FUNCTION_BLOCK "ifbHMISelectBLK"
{ S7_Optimized_Access := 'TRUE' }
VERSION : 0.1
   VAR
      edge : Array[0..50] of Bool;
   END_VAR

   VAR_TEMP
      blockSelected : Int;
      arrChildIndex : Array[0..50] of Int;
      tempEdge : Bool;
   END_VAR


BEGIN
NETWORK
TITLE = Get the selected BLK
//------------------------------------------------------------------------//
// Get the BLK index number selected by the user when they clicked the    //
// faceplate BLK target:                                                  //
//------------------------------------------------------------------------//
      L "dbHMIInterfaceBLK".block.blockSelected;
      T #blockSelected;

NETWORK
TITLE =
      A(;
      L #blockSelected;
      L 1134;
      ==I;
      );
      FP #edge[0];
      = #tempEdge;
      JCN out1;

      A "idbEMA1".f[0].p.read.mc.modeAUTO;
      R "dbHMIInterfaceBLK".block.manual;

      A "idbEMA1".f[0].p.read.mc.modeMANUAL;
      S "dbHMIInterfaceBLK".block.manual;

out1:      NOP 0;

NETWORK
TITLE = EA1010 M1 Vessel Agitator
//------------------------------------------------------------------------//
// Check if this BLK instance is selected:                                //
//------------------------------------------------------------------------//
      A(;
      L #blockSelected;
      L 1134;
      ==I;
      );

      JCN _not_EA1010;
      AN #tempEdge;
      CALL "fcHMIInterfaceBLK"
      (  mcr                         := "idbEMA1".f[0].p.read.mc ,
         mcw                         := "idbEMA1".f[0].p.write.mc ,
         bmc                         := "idbEMA1".f[0].p.read.bmc
      );

NETWORK
TITLE = Transfer the child state values and errors to the interface array
//------------------------------------------------------------------------//
// Transfer the child states and if they have any error condition:        //
//------------------------------------------------------------------------//
      L 0        ;// SIC_AGIT SIC1
      T #arrChildIndex[1];
      L "idbSIC1".f[#arrChildIndex[1]].p.read.mc.STATE;
      T "dbHMIInterfaceBLK".block.arrChildState[1];
      A "idbSIC1".f[#arrChildIndex[1]].p.read.mc.ERROR;
      = "dbHMIInterfaceBLK".block.arrChildError[1];
      A "idbSIC1".f[#arrChildIndex[1]].p.read.mc.INTERLOCK;
      = "dbHMIInterfaceBLK".block.arrChildInterlock[1];

NETWORK
TITLE = Transfer the parameter values to the interface arrays
//------------------------------------------------------------------------//
// Transfer the parameter values:                                         //
//------------------------------------------------------------------------//
      AN "dbHMIInterfaceBLK".block.manual;
      JCN _manual_EA1010;
      A "idbEMA1".f[0].p.read.AGIT_RUNNING;
      = "dbHMIInterfaceBLK".block.arrBool[1];
      A "idbEMA1".f[0].p.read.AGIT_STOPPED;
      = "dbHMIInterfaceBLK".block.arrBool[2];
      A "idbEMA1".f[0].p.read.RESETRUNTIMER;
      = "dbHMIInterfaceBLK".block.arrBool[3];
      L "idbEMA1".f[0].p.read.ACUMTIMEH;
      T "dbHMIInterfaceBLK".block.arrInt[1];
      L "idbEMA1".f[0].p.read.ACUMTIMEM;
      T "dbHMIInterfaceBLK".block.arrInt[2];
      L "idbEMA1".f[0].p.read.ACUMTIMES;
      T "dbHMIInterfaceBLK".block.arrInt[3];
      L "idbEMA1".f[0].p.write.RUNTIME_H;
      T "dbHMIInterfaceBLK".block.arrInt[4];
      L "idbEMA1".f[0].p.write.RUNTIME_M;
      T "dbHMIInterfaceBLK".block.arrInt[5];
      L "idbEMA1".f[0].p.write.RUNTIME_S;
      T "dbHMIInterfaceBLK".block.arrInt[6];
      L "idbEMA1".f[0].p.write.SETPOINT;
      T "dbHMIInterfaceBLK".block.arrReal[1];
_manual_EA1010:      NOP 0;

NETWORK
TITLE = Transfer the parameter values to the interface arrays
//------------------------------------------------------------------------//
// Transfer the parameter values:                                         //
//------------------------------------------------------------------------//
      A "dbHMIInterfaceBLK".block.manual;
      JCN _auto_EA1010;
      A "dbHMIInterfaceBLK".block.arrBool[1];
      = "idbEMA1".f[0].p.read.AGIT_RUNNING;
      A "dbHMIInterfaceBLK".block.arrBool[2];
      = "idbEMA1".f[0].p.read.AGIT_STOPPED;
      A "dbHMIInterfaceBLK".block.arrBool[3];
      = "idbEMA1".f[0].p.read.RESETRUNTIMER;
      L "dbHMIInterfaceBLK".block.arrInt[1];
      T "idbEMA1".f[0].p.read.ACUMTIMEH;
      L "dbHMIInterfaceBLK".block.arrInt[2];
      T "idbEMA1".f[0].p.read.ACUMTIMEM;
      L "dbHMIInterfaceBLK".block.arrInt[3];
      T "idbEMA1".f[0].p.read.ACUMTIMES;
      L "dbHMIInterfaceBLK".block.arrInt[4];
      T "idbEMA1".f[0].p.write.RUNTIME_H;
      L "dbHMIInterfaceBLK".block.arrInt[5];
      T "idbEMA1".f[0].p.write.RUNTIME_M;
      L "dbHMIInterfaceBLK".block.arrInt[6];
      T "idbEMA1".f[0].p.write.RUNTIME_S;
      L "dbHMIInterfaceBLK".block.arrReal[1];
      T "idbEMA1".f[0].p.write.SETPOINT;
_auto_EA1010:      NOP 0;

_not_EA1010:      NOP 0;

NETWORK
TITLE = EC1001 M1 LP CA and HP CA supply and Vacuum and Vent
//------------------------------------------------------------------------//
// Check if this BLK instance is selected:                                //
//------------------------------------------------------------------------//
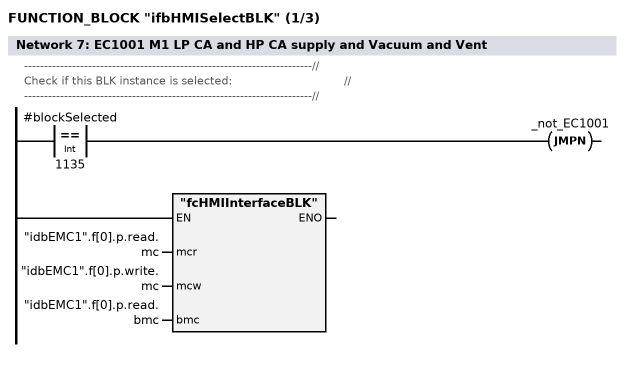
      A(;
      L #blockSelected;
      L 1135;
      ==I;
      );
      JCN _not_EC1001;

      CALL "fcHMIInterfaceBLK"
      (  mcr                         := "idbEMC1".f[0].p.read.mc ,
         mcw                         := "idbEMC1".f[0].p.write.mc ,
         bmc                         := "idbEMC1".f[0].p.read.bmc
      );

NETWORK
TITLE = Transfer the child state values and errors to the interface array
//------------------------------------------------------------------------//
// Transfer the child states and if they have any error condition:        //
//------------------------------------------------------------------------//
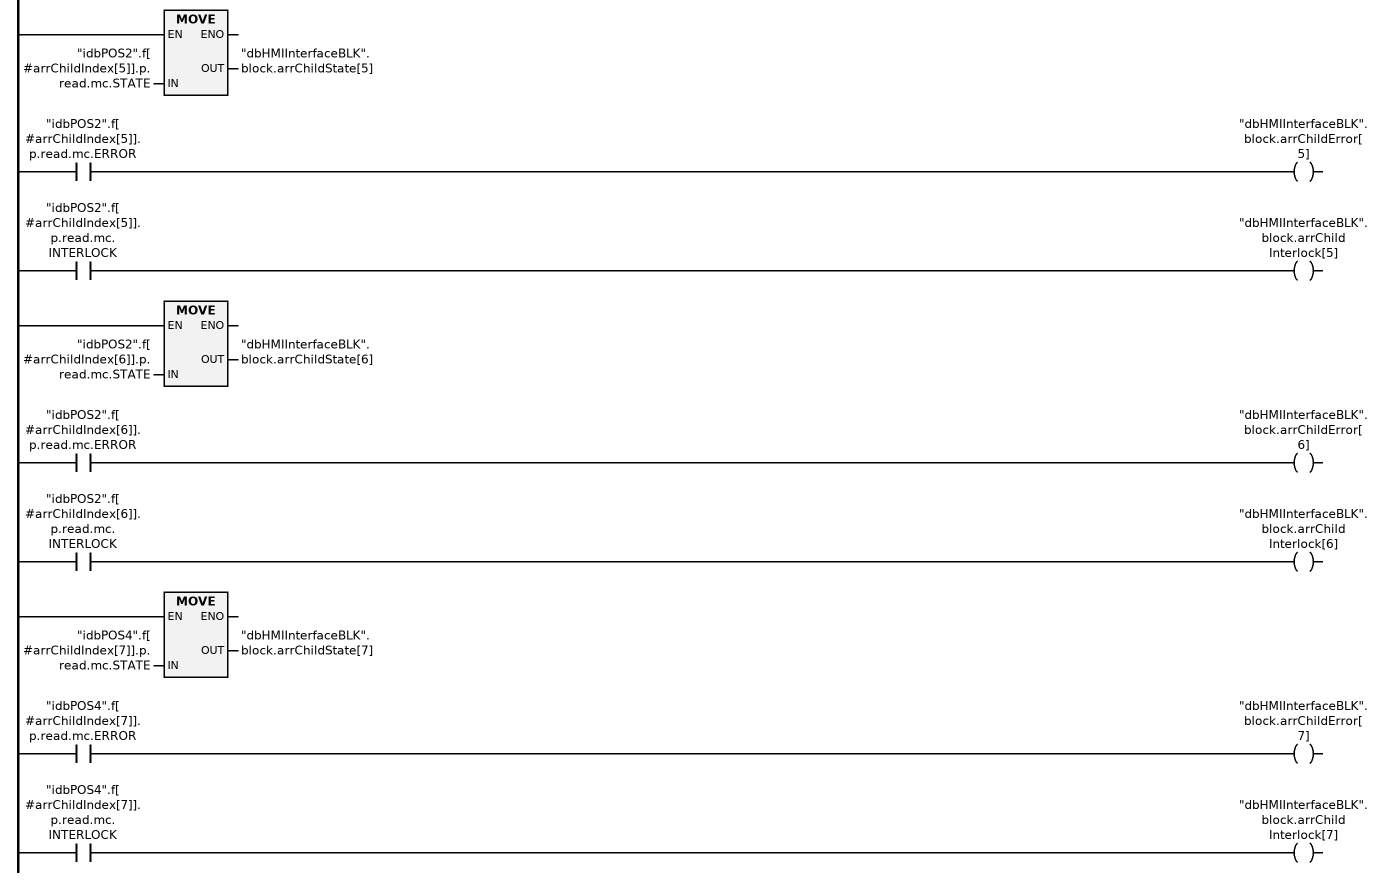
      L 0        ;// PC_VESSEL PC1
      T #arrChildIndex[1];
      L 0        ;// PI_VESSEL PI1
      T #arrChildIndex[2];
      L 1        ;// POS_HPCA POS2
      T #arrChildIndex[3];
      L 2        ;// POS_LPCA POS2
      T #arrChildIndex[4];
      L 3        ;// POS_VACUUM POS2
      T #arrChildIndex[5];
      L 0        ;// POS_VENT POS2
      T #arrChildIndex[6];
      L 0        ;// POS_DRAIN POS4
      T #arrChildIndex[7];
      L "idbPC1".f[#arrChildIndex[1]].p.read.mc.STATE;
      T "dbHMIInterfaceBLK".block.arrChildState[1];
      A "idbPC1".f[#arrChildIndex[1]].p.read.mc.ERROR;
      = "dbHMIInterfaceBLK".block.arrChildError[1];
      A "idbPC1".f[#arrChildIndex[1]].p.read.mc.INTERLOCK;
      = "dbHMIInterfaceBLK".block.arrChildInterlock[1];
      L "idbPI1".f[#arrChildIndex[2]].p.read.mc.STATE;
      T "dbHMIInterfaceBLK".block.arrChildState[2];
      A "idbPI1".f[#arrChildIndex[2]].p.read.mc.ERROR;
      = "dbHMIInterfaceBLK".block.arrChildError[2];
      A "idbPI1".f[#arrChildIndex[2]].p.read.mc.INTERLOCK;
      = "dbHMIInterfaceBLK".block.arrChildInterlock[2];
      L "idbPOS2".f[#arrChildIndex[3]].p.read.mc.STATE;
      T "dbHMIInterfaceBLK".block.arrChildState[3];
      A "idbPOS2".f[#arrChildIndex[3]].p.read.mc.ERROR;
      = "dbHMIInterfaceBLK".block.arrChildError[3];
      A "idbPOS2".f[#arrChildIndex[3]].p.read.mc.INTERLOCK;
      = "dbHMIInterfaceBLK".block.arrChildInterlock[3];
      L "idbPOS2".f[#arrChildIndex[4]].p.read.mc.STATE;
      T "dbHMIInterfaceBLK".block.arrChildState[4];
      A "idbPOS2".f[#arrChildIndex[4]].p.read.mc.ERROR;
      = "dbHMIInterfaceBLK".block.arrChildError[4];
      A "idbPOS2".f[#arrChildIndex[4]].p.read.mc.INTERLOCK;
      = "dbHMIInterfaceBLK".block.arrChildInterlock[4];
      L "idbPOS2".f[#arrChildIndex[5]].p.read.mc.STATE;
      T "dbHMIInterfaceBLK".block.arrChildState[5];
      A "idbPOS2".f[#arrChildIndex[5]].p.read.mc.ERROR;
      = "dbHMIInterfaceBLK".block.arrChildError[5];
      A "idbPOS2".f[#arrChildIndex[5]].p.read.mc.INTERLOCK;
      = "dbHMIInterfaceBLK".block.arrChildInterlock[5];
      L "idbPOS2".f[#arrChildIndex[6]].p.read.mc.STATE;
      T "dbHMIInterfaceBLK".block.arrChildState[6];
      A "idbPOS2".f[#arrChildIndex[6]].p.read.mc.ERROR;
      = "dbHMIInterfaceBLK".block.arrChildError[6];
      A "idbPOS2".f[#arrChildIndex[6]].p.read.mc.INTERLOCK;
      = "dbHMIInterfaceBLK".block.arrChildInterlock[6];
      L "idbPOS4".f[#arrChildIndex[7]].p.read.mc.STATE;
      T "dbHMIInterfaceBLK".block.arrChildState[7];
      A "idbPOS4".f[#arrChildIndex[7]].p.read.mc.ERROR;
      = "dbHMIInterfaceBLK".block.arrChildError[7];
      A "idbPOS4".f[#arrChildIndex[7]].p.read.mc.INTERLOCK;
      = "dbHMIInterfaceBLK".block.arrChildInterlock[7];

NETWORK
TITLE = Transfer the parameter values to the interface arrays
//------------------------------------------------------------------------//
// Transfer the parameter values:                                         //
//------------------------------------------------------------------------//
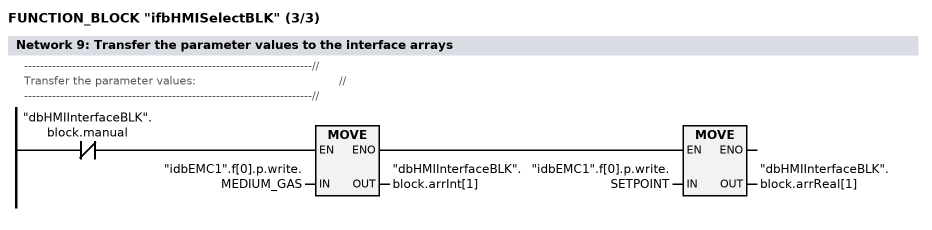
      AN "dbHMIInterfaceBLK".block.manual;
      JCN _manual_EC1001;
      L "idbEMC1".f[0].p.write.MEDIUM_GAS;
      T "dbHMIInterfaceBLK".block.arrInt[1];
      L "idbEMC1".f[0].p.write.SETPOINT;
      T "dbHMIInterfaceBLK".block.arrReal[1];
_manual_EC1001:      NOP 0;

NETWORK
TITLE = Transfer the parameter values to the interface arrays
//------------------------------------------------------------------------//
// Transfer the parameter values:                                         //
//------------------------------------------------------------------------//
      A "dbHMIInterfaceBLK".block.manual;
      JCN _auto_EC1001;
      L "dbHMIInterfaceBLK".block.arrInt[1];
      T "idbEMC1".f[0].p.write.MEDIUM_GAS;
      L "dbHMIInterfaceBLK".block.arrReal[1];
      T "idbEMC1".f[0].p.write.SETPOINT;
_auto_EC1001:      NOP 0;

_not_EC1001:      NOP 0;

NETWORK
TITLE = EC1002 M1 WFI and PS supply plus PW and PS supply
//------------------------------------------------------------------------//
// Check if this BLK instance is selected:                                //
//------------------------------------------------------------------------//
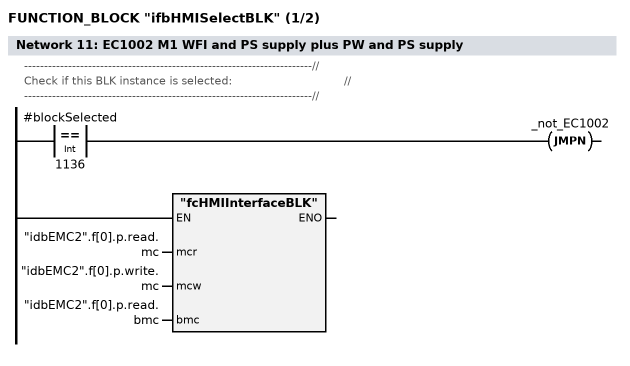
      A(;
      L #blockSelected;
      L 1136;
      ==I;
      );
      JCN _not_EC1002;

      CALL "fcHMIInterfaceBLK"
      (  mcr                         := "idbEMC2".f[0].p.read.mc ,
         mcw                         := "idbEMC2".f[0].p.write.mc ,
         bmc                         := "idbEMC2".f[0].p.read.bmc
      );

NETWORK
TITLE = Transfer the child state values and errors to the interface array
//------------------------------------------------------------------------//
// Transfer the child states and if they have any error condition:        //
//------------------------------------------------------------------------//
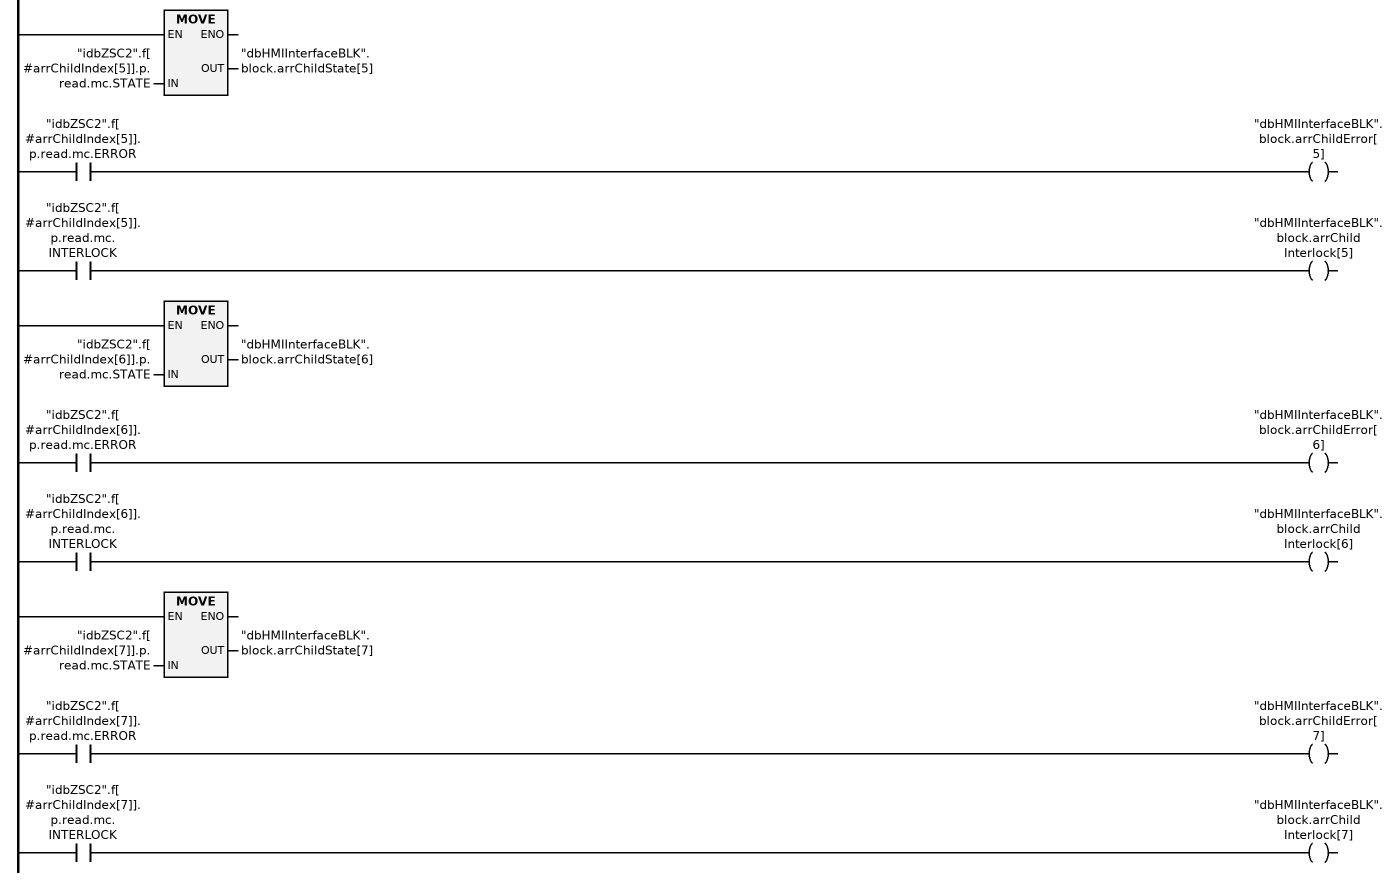
      L 5        ;// POS_PSPW POS2
      T #arrChildIndex[1];
      L 4        ;// POS_PSWFI POS2
      T #arrChildIndex[2];
      L 29        ;// POS_PW POS4
      T #arrChildIndex[3];
      L 28        ;// POS_WFI POS4
      T #arrChildIndex[4];
      L 2        ;// ZSC_FPINLET ZSC2
      T #arrChildIndex[5];
      L 1        ;// ZSC_FPPW ZSC2
      T #arrChildIndex[6];
      L 0        ;// ZSC_FPWFI ZSC2
      T #arrChildIndex[7];
      L "idbPOS2".f[#arrChildIndex[1]].p.read.mc.STATE;
      T "dbHMIInterfaceBLK".block.arrChildState[1];
      A "idbPOS2".f[#arrChildIndex[1]].p.read.mc.ERROR;
      = "dbHMIInterfaceBLK".block.arrChildError[1];
      A "idbPOS2".f[#arrChildIndex[1]].p.read.mc.INTERLOCK;
      = "dbHMIInterfaceBLK".block.arrChildInterlock[1];
      L "idbPOS2".f[#arrChildIndex[2]].p.read.mc.STATE;
      T "dbHMIInterfaceBLK".block.arrChildState[2];
      A "idbPOS2".f[#arrChildIndex[2]].p.read.mc.ERROR;
      = "dbHMIInterfaceBLK".block.arrChildError[2];
      A "idbPOS2".f[#arrChildIndex[2]].p.read.mc.INTERLOCK;
      = "dbHMIInterfaceBLK".block.arrChildInterlock[2];
      L "idbPOS4".f[#arrChildIndex[3]].p.read.mc.STATE;
      T "dbHMIInterfaceBLK".block.arrChildState[3];
      A "idbPOS4".f[#arrChildIndex[3]].p.read.mc.ERROR;
      = "dbHMIInterfaceBLK".block.arrChildError[3];
      A "idbPOS4".f[#arrChildIndex[3]].p.read.mc.INTERLOCK;
      = "dbHMIInterfaceBLK".block.arrChildInterlock[3];
      L "idbPOS4".f[#arrChildIndex[4]].p.read.mc.STATE;
      T "dbHMIInterfaceBLK".block.arrChildState[4];
      A "idbPOS4".f[#arrChildIndex[4]].p.read.mc.ERROR;
      = "dbHMIInterfaceBLK".block.arrChildError[4];
      A "idbPOS4".f[#arrChildIndex[4]].p.read.mc.INTERLOCK;
      = "dbHMIInterfaceBLK".block.arrChildInterlock[4];
      L "idbZSC2".f[#arrChildIndex[5]].p.read.mc.STATE;
      T "dbHMIInterfaceBLK".block.arrChildState[5];
      A "idbZSC2".f[#arrChildIndex[5]].p.read.mc.ERROR;
      = "dbHMIInterfaceBLK".block.arrChildError[5];
      A "idbZSC2".f[#arrChildIndex[5]].p.read.mc.INTERLOCK;
      = "dbHMIInterfaceBLK".block.arrChildInterlock[5];
      L "idbZSC2".f[#arrChildIndex[6]].p.read.mc.STATE;
      T "dbHMIInterfaceBLK".block.arrChildState[6];
      A "idbZSC2".f[#arrChildIndex[6]].p.read.mc.ERROR;
      = "dbHMIInterfaceBLK".block.arrChildError[6];
      A "idbZSC2".f[#arrChildIndex[6]].p.read.mc.INTERLOCK;
      = "dbHMIInterfaceBLK".block.arrChildInterlock[6];
      L "idbZSC2".f[#arrChildIndex[7]].p.read.mc.STATE;
      T "dbHMIInterfaceBLK".block.arrChildState[7];
      A "idbZSC2".f[#arrChildIndex[7]].p.read.mc.ERROR;
      = "dbHMIInterfaceBLK".block.arrChildError[7];
      A "idbZSC2".f[#arrChildIndex[7]].p.read.mc.INTERLOCK;
      = "dbHMIInterfaceBLK".block.arrChildInterlock[7];

NETWORK
TITLE = Transfer the parameter values to the interface arrays
//------------------------------------------------------------------------//
// Transfer the parameter values:                                         //
//------------------------------------------------------------------------//
      AN "dbHMIInterfaceBLK".block.manual;
      JCN _manual_EC1002;
      A "idbEMC2".f[0].p.read.MASS_READY;
      = "dbHMIInterfaceBLK".block.arrBool[1];
      L "idbEMC2".f[0].p.write.MEDIUM_LIQUID;
      T "dbHMIInterfaceBLK".block.arrInt[1];
      L "idbEMC2".f[0].p.read.MASS_ACTUAL;
      T "dbHMIInterfaceBLK".block.arrReal[1];
      L "idbEMC2".f[0].p.read.MASS_FINAL;
      T "dbHMIInterfaceBLK".block.arrReal[2];
      L "idbEMC2".f[0].p.read.MASS_INITIAL;
      T "dbHMIInterfaceBLK".block.arrReal[3];
      L "idbEMC2".f[0].p.write.MASS_CHARGE;
      T "dbHMIInterfaceBLK".block.arrReal[4];
      L "idbEMC2".f[0].p.write.RUNTIME;
      T "dbHMIInterfaceBLK".block.arrTime[1];
      L "idbEMC2".f[0].p.write.TIMEOUT;
      T "dbHMIInterfaceBLK".block.arrTime[2];
_manual_EC1002:      NOP 0;

NETWORK
TITLE = Transfer the parameter values to the interface arrays
//------------------------------------------------------------------------//
// Transfer the parameter values:                                         //
//------------------------------------------------------------------------//
      A "dbHMIInterfaceBLK".block.manual;
      JCN _auto_EC1002;
      A "dbHMIInterfaceBLK".block.arrBool[1];
      = "idbEMC2".f[0].p.read.MASS_READY;
      L "dbHMIInterfaceBLK".block.arrInt[1];
      T "idbEMC2".f[0].p.write.MEDIUM_LIQUID;
      L "dbHMIInterfaceBLK".block.arrReal[1];
      T "idbEMC2".f[0].p.read.MASS_ACTUAL;
      L "dbHMIInterfaceBLK".block.arrReal[2];
      T "idbEMC2".f[0].p.read.MASS_FINAL;
      L "dbHMIInterfaceBLK".block.arrReal[3];
      T "idbEMC2".f[0].p.read.MASS_INITIAL;
      L "dbHMIInterfaceBLK".block.arrReal[4];
      T "idbEMC2".f[0].p.write.MASS_CHARGE;
      L "dbHMIInterfaceBLK".block.arrTime[1];
      T "idbEMC2".f[0].p.write.RUNTIME;
      L "dbHMIInterfaceBLK".block.arrTime[2];
      T "idbEMC2".f[0].p.write.TIMEOUT;
_auto_EC1002:      NOP 0;

_not_EC1002:      NOP 0;

NETWORK
TITLE = EC3001 S1 LP CA and HP CA supply and Vacuum and Vent
//------------------------------------------------------------------------//
// Check if this BLK instance is selected:                                //
//------------------------------------------------------------------------//
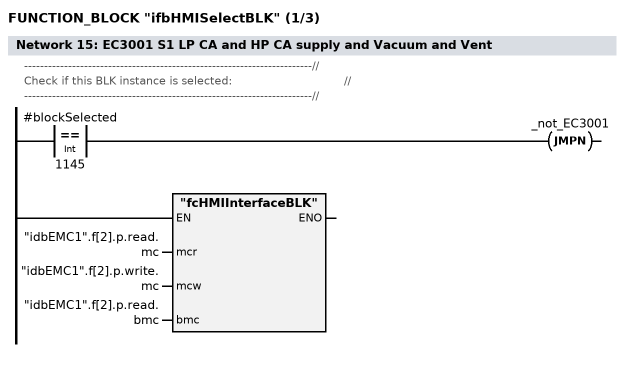
      A(;
      L #blockSelected;
      L 1145;
      ==I;
      );
      JCN _not_EC3001;

      CALL "fcHMIInterfaceBLK"
      (  mcr                         := "idbEMC1".f[2].p.read.mc ,
         mcw                         := "idbEMC1".f[2].p.write.mc ,
         bmc                         := "idbEMC1".f[2].p.read.bmc
      );

NETWORK
TITLE = Transfer the child state values and errors to the interface array
//------------------------------------------------------------------------//
// Transfer the child states and if they have any error condition:        //
//------------------------------------------------------------------------//
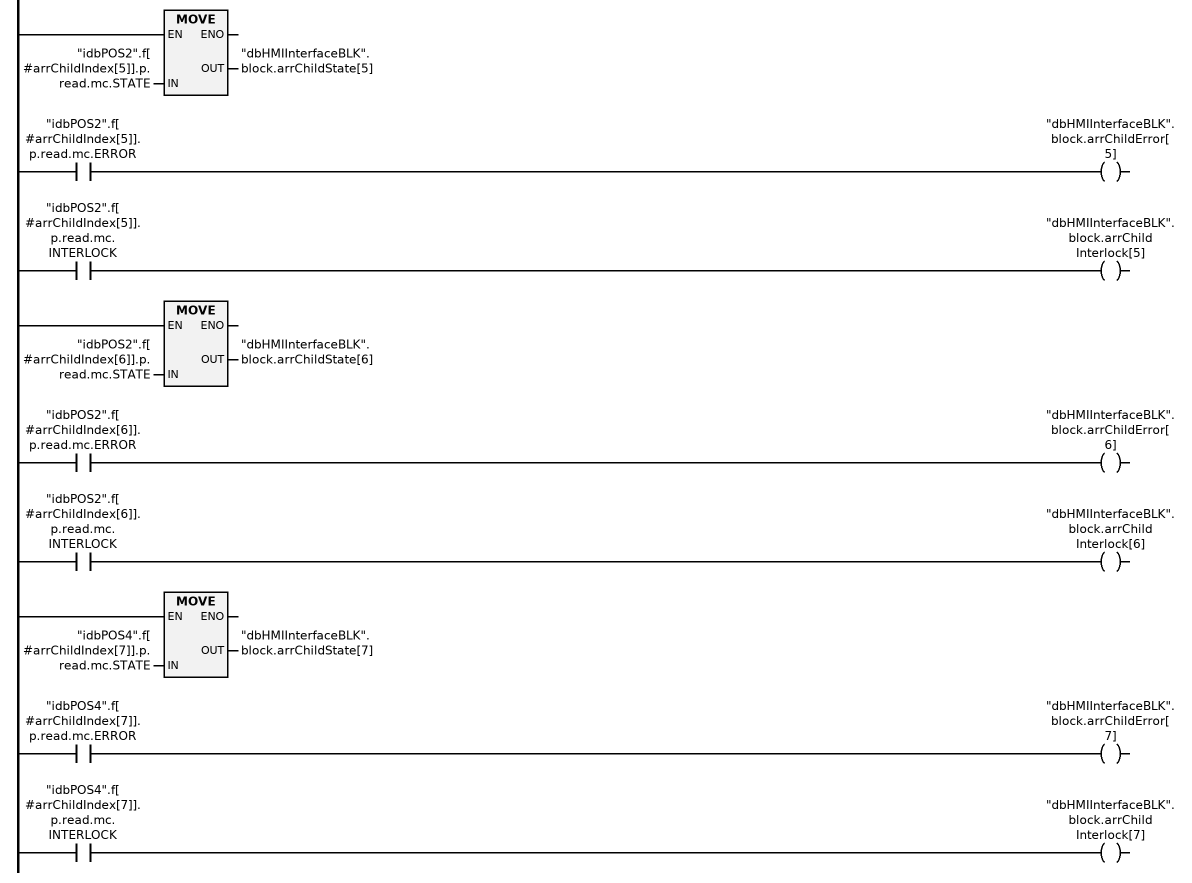
      L 2        ;// PC_VESSEL PC1
      T #arrChildIndex[1];
      L 2        ;// PI_VESSEL PI1
      T #arrChildIndex[2];
      L 27        ;// POS_HPCA POS2
      T #arrChildIndex[3];
      L 28        ;// POS_LPCA POS2
      T #arrChildIndex[4];
      L 29        ;// POS_VACUUM POS2
      T #arrChildIndex[5];
      L 26        ;// POS_VENT POS2
      T #arrChildIndex[6];
      L 16        ;// POS_DRAIN POS4
      T #arrChildIndex[7];
      L "idbPC1".f[#arrChildIndex[1]].p.read.mc.STATE;
      T "dbHMIInterfaceBLK".block.arrChildState[1];
      A "idbPC1".f[#arrChildIndex[1]].p.read.mc.ERROR;
      = "dbHMIInterfaceBLK".block.arrChildError[1];
      A "idbPC1".f[#arrChildIndex[1]].p.read.mc.INTERLOCK;
      = "dbHMIInterfaceBLK".block.arrChildInterlock[1];
      L "idbPI1".f[#arrChildIndex[2]].p.read.mc.STATE;
      T "dbHMIInterfaceBLK".block.arrChildState[2];
      A "idbPI1".f[#arrChildIndex[2]].p.read.mc.ERROR;
      = "dbHMIInterfaceBLK".block.arrChildError[2];
      A "idbPI1".f[#arrChildIndex[2]].p.read.mc.INTERLOCK;
      = "dbHMIInterfaceBLK".block.arrChildInterlock[2];
      L "idbPOS2".f[#arrChildIndex[3]].p.read.mc.STATE;
      T "dbHMIInterfaceBLK".block.arrChildState[3];
      A "idbPOS2".f[#arrChildIndex[3]].p.read.mc.ERROR;
      = "dbHMIInterfaceBLK".block.arrChildError[3];
      A "idbPOS2".f[#arrChildIndex[3]].p.read.mc.INTERLOCK;
      = "dbHMIInterfaceBLK".block.arrChildInterlock[3];
      L "idbPOS2".f[#arrChildIndex[4]].p.read.mc.STATE;
      T "dbHMIInterfaceBLK".block.arrChildState[4];
      A "idbPOS2".f[#arrChildIndex[4]].p.read.mc.ERROR;
      = "dbHMIInterfaceBLK".block.arrChildError[4];
      A "idbPOS2".f[#arrChildIndex[4]].p.read.mc.INTERLOCK;
      = "dbHMIInterfaceBLK".block.arrChildInterlock[4];
      L "idbPOS2".f[#arrChildIndex[5]].p.read.mc.STATE;
      T "dbHMIInterfaceBLK".block.arrChildState[5];
      A "idbPOS2".f[#arrChildIndex[5]].p.read.mc.ERROR;
      = "dbHMIInterfaceBLK".block.arrChildError[5];
      A "idbPOS2".f[#arrChildIndex[5]].p.read.mc.INTERLOCK;
      = "dbHMIInterfaceBLK".block.arrChildInterlock[5];
      L "idbPOS2".f[#arrChildIndex[6]].p.read.mc.STATE;
      T "dbHMIInterfaceBLK".block.arrChildState[6];
      A "idbPOS2".f[#arrChildIndex[6]].p.read.mc.ERROR;
      = "dbHMIInterfaceBLK".block.arrChildError[6];
      A "idbPOS2".f[#arrChildIndex[6]].p.read.mc.INTERLOCK;
      = "dbHMIInterfaceBLK".block.arrChildInterlock[6];
      L "idbPOS4".f[#arrChildIndex[7]].p.read.mc.STATE;
      T "dbHMIInterfaceBLK".block.arrChildState[7];
      A "idbPOS4".f[#arrChildIndex[7]].p.read.mc.ERROR;
      = "dbHMIInterfaceBLK".block.arrChildError[7];
      A "idbPOS4".f[#arrChildIndex[7]].p.read.mc.INTERLOCK;
      = "dbHMIInterfaceBLK".block.arrChildInterlock[7];

NETWORK
TITLE = Transfer the parameter values to the interface arrays
//------------------------------------------------------------------------//
// Transfer the parameter values:                                         //
//------------------------------------------------------------------------//
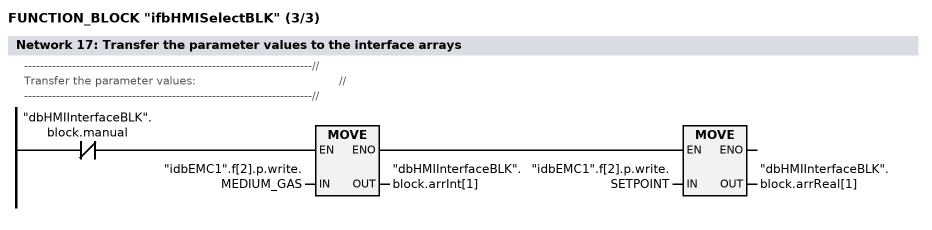
      AN "dbHMIInterfaceBLK".block.manual;
      JCN _manual_EC3001;
      L "idbEMC1".f[2].p.write.MEDIUM_GAS;
      T "dbHMIInterfaceBLK".block.arrInt[1];
      L "idbEMC1".f[2].p.write.SETPOINT;
      T "dbHMIInterfaceBLK".block.arrReal[1];
_manual_EC3001:      NOP 0;

NETWORK
TITLE = Transfer the parameter values to the interface arrays
//------------------------------------------------------------------------//
// Transfer the parameter values:                                         //
//------------------------------------------------------------------------//
      A "dbHMIInterfaceBLK".block.manual;
      JCN _auto_EC3001;
      L "dbHMIInterfaceBLK".block.arrInt[1];
      T "idbEMC1".f[2].p.write.MEDIUM_GAS;
      L "dbHMIInterfaceBLK".block.arrReal[1];
      T "idbEMC1".f[2].p.write.SETPOINT;
_auto_EC3001:      NOP 0;

_not_EC3001:      NOP 0;

NETWORK
TITLE = EC3002 S1 WFI and PS supply plus PW and PS supply
//------------------------------------------------------------------------//
// Check if this BLK instance is selected:                                //
//------------------------------------------------------------------------//
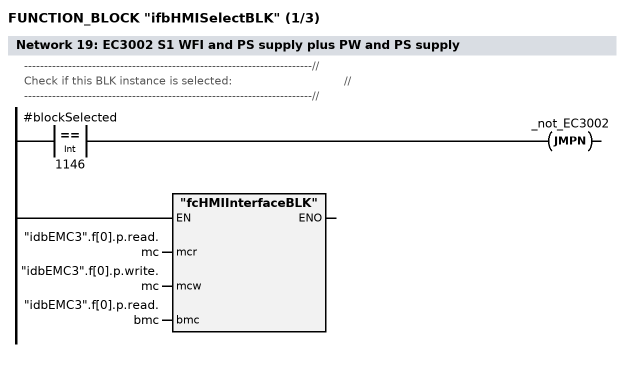
      A(;
      L #blockSelected;
      L 1146;
      ==I;
      );
      JCN _not_EC3002;

      CALL "fcHMIInterfaceBLK"
      (  mcr                         := "idbEMC3".f[0].p.read.mc ,
         mcw                         := "idbEMC3".f[0].p.write.mc ,
         bmc                         := "idbEMC3".f[0].p.read.bmc
      );

NETWORK
TITLE = Transfer the child state values and errors to the interface array
//------------------------------------------------------------------------//
// Transfer the child states and if they have any error condition:        //
//------------------------------------------------------------------------//
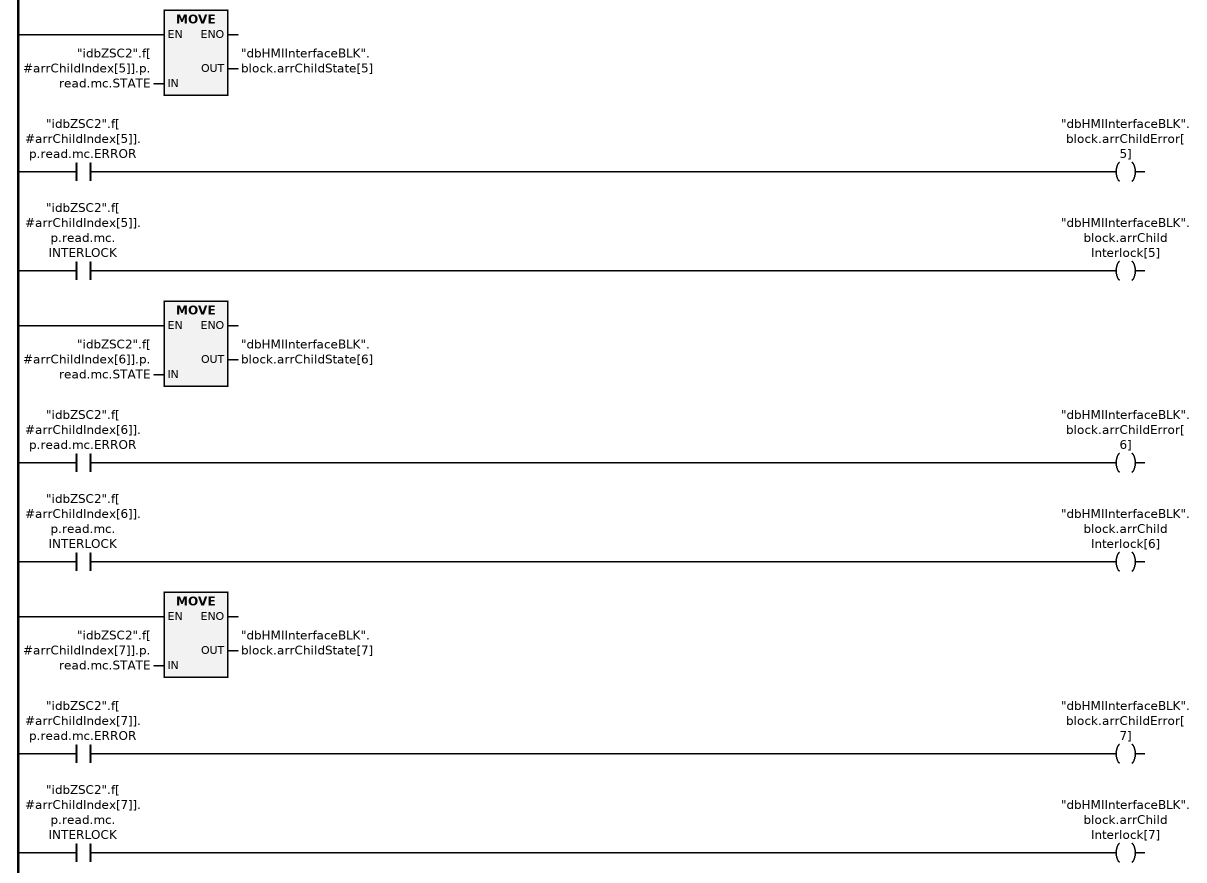
      L 31        ;// POS_PSPW POS2
      T #arrChildIndex[1];
      L 30        ;// POS_PSWFI POS2
      T #arrChildIndex[2];
      L 33        ;// POS_PW POS4
      T #arrChildIndex[3];
      L 32        ;// POS_WFI POS4
      T #arrChildIndex[4];
      L 16        ;// ZSC_FPINLET ZSC2
      T #arrChildIndex[5];
      L 15        ;// ZSC_FPPW ZSC2
      T #arrChildIndex[6];
      L 14        ;// ZSC_FPWFI ZSC2
      T #arrChildIndex[7];
      L "idbPOS2".f[#arrChildIndex[1]].p.read.mc.STATE;
      T "dbHMIInterfaceBLK".block.arrChildState[1];
      A "idbPOS2".f[#arrChildIndex[1]].p.read.mc.ERROR;
      = "dbHMIInterfaceBLK".block.arrChildError[1];
      A "idbPOS2".f[#arrChildIndex[1]].p.read.mc.INTERLOCK;
      = "dbHMIInterfaceBLK".block.arrChildInterlock[1];
      L "idbPOS2".f[#arrChildIndex[2]].p.read.mc.STATE;
      T "dbHMIInterfaceBLK".block.arrChildState[2];
      A "idbPOS2".f[#arrChildIndex[2]].p.read.mc.ERROR;
      = "dbHMIInterfaceBLK".block.arrChildError[2];
      A "idbPOS2".f[#arrChildIndex[2]].p.read.mc.INTERLOCK;
      = "dbHMIInterfaceBLK".block.arrChildInterlock[2];
      L "idbPOS4".f[#arrChildIndex[3]].p.read.mc.STATE;
      T "dbHMIInterfaceBLK".block.arrChildState[3];
      A "idbPOS4".f[#arrChildIndex[3]].p.read.mc.ERROR;
      = "dbHMIInterfaceBLK".block.arrChildError[3];
      A "idbPOS4".f[#arrChildIndex[3]].p.read.mc.INTERLOCK;
      = "dbHMIInterfaceBLK".block.arrChildInterlock[3];
      L "idbPOS4".f[#arrChildIndex[4]].p.read.mc.STATE;
      T "dbHMIInterfaceBLK".block.arrChildState[4];
      A "idbPOS4".f[#arrChildIndex[4]].p.read.mc.ERROR;
      = "dbHMIInterfaceBLK".block.arrChildError[4];
      A "idbPOS4".f[#arrChildIndex[4]].p.read.mc.INTERLOCK;
      = "dbHMIInterfaceBLK".block.arrChildInterlock[4];
      L "idbZSC2".f[#arrChildIndex[5]].p.read.mc.STATE;
      T "dbHMIInterfaceBLK".block.arrChildState[5];
      A "idbZSC2".f[#arrChildIndex[5]].p.read.mc.ERROR;
      = "dbHMIInterfaceBLK".block.arrChildError[5];
      A "idbZSC2".f[#arrChildIndex[5]].p.read.mc.INTERLOCK;
      = "dbHMIInterfaceBLK".block.arrChildInterlock[5];
      L "idbZSC2".f[#arrChildIndex[6]].p.read.mc.STATE;
      T "dbHMIInterfaceBLK".block.arrChildState[6];
      A "idbZSC2".f[#arrChildIndex[6]].p.read.mc.ERROR;
      = "dbHMIInterfaceBLK".block.arrChildError[6];
      A "idbZSC2".f[#arrChildIndex[6]].p.read.mc.INTERLOCK;
      = "dbHMIInterfaceBLK".block.arrChildInterlock[6];
      L "idbZSC2".f[#arrChildIndex[7]].p.read.mc.STATE;
      T "dbHMIInterfaceBLK".block.arrChildState[7];
      A "idbZSC2".f[#arrChildIndex[7]].p.read.mc.ERROR;
      = "dbHMIInterfaceBLK".block.arrChildError[7];
      A "idbZSC2".f[#arrChildIndex[7]].p.read.mc.INTERLOCK;
      = "dbHMIInterfaceBLK".block.arrChildInterlock[7];

NETWORK
TITLE = Transfer the parameter values to the interface arrays
//------------------------------------------------------------------------//
// Transfer the parameter values:                                         //
//------------------------------------------------------------------------//
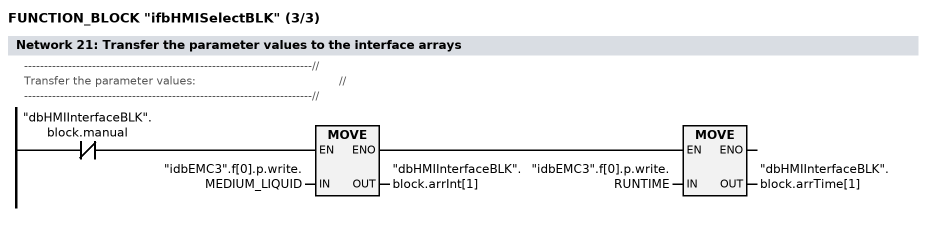
      AN "dbHMIInterfaceBLK".block.manual;
      JCN _manual_EC3002;
      L "idbEMC3".f[0].p.write.MEDIUM_LIQUID;
      T "dbHMIInterfaceBLK".block.arrInt[1];
      L "idbEMC3".f[0].p.write.RUNTIME;
      T "dbHMIInterfaceBLK".block.arrTime[1];
_manual_EC3002:      NOP 0;

NETWORK
TITLE = Transfer the parameter values to the interface arrays
//------------------------------------------------------------------------//
// Transfer the parameter values:                                         //
//------------------------------------------------------------------------//
      A "dbHMIInterfaceBLK".block.manual;
      JCN _auto_EC3002;
      L "dbHMIInterfaceBLK".block.arrInt[1];
      T "idbEMC3".f[0].p.write.MEDIUM_LIQUID;
      L "dbHMIInterfaceBLK".block.arrTime[1];
      T "idbEMC3".f[0].p.write.RUNTIME;
_auto_EC3002:      NOP 0;

_not_EC3002:      NOP 0;

NETWORK
TITLE = EG1005 M1 gas filter heating and drain valve and temperature indicator
//------------------------------------------------------------------------//
// Check if this BLK instance is selected:                                //
//------------------------------------------------------------------------//
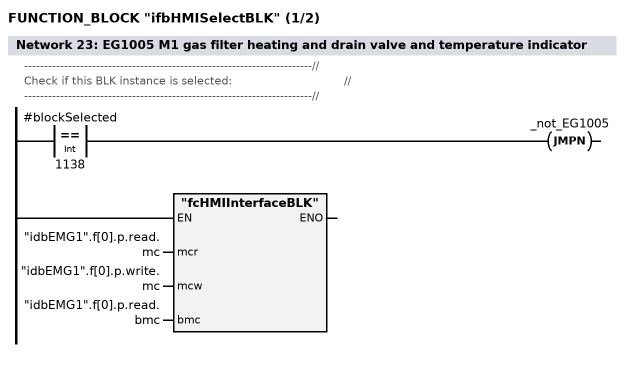
      A(;
      L #blockSelected;
      L 1138;
      ==I;
      );
      JCN _not_EG1005;

      CALL "fcHMIInterfaceBLK"
      (  mcr                         := "idbEMG1".f[0].p.read.mc ,
         mcw                         := "idbEMG1".f[0].p.write.mc ,
         bmc                         := "idbEMG1".f[0].p.read.bmc
      );

NETWORK
TITLE = Transfer the child state values and errors to the interface array
//------------------------------------------------------------------------//
// Transfer the child states and if they have any error condition:        //
//------------------------------------------------------------------------//
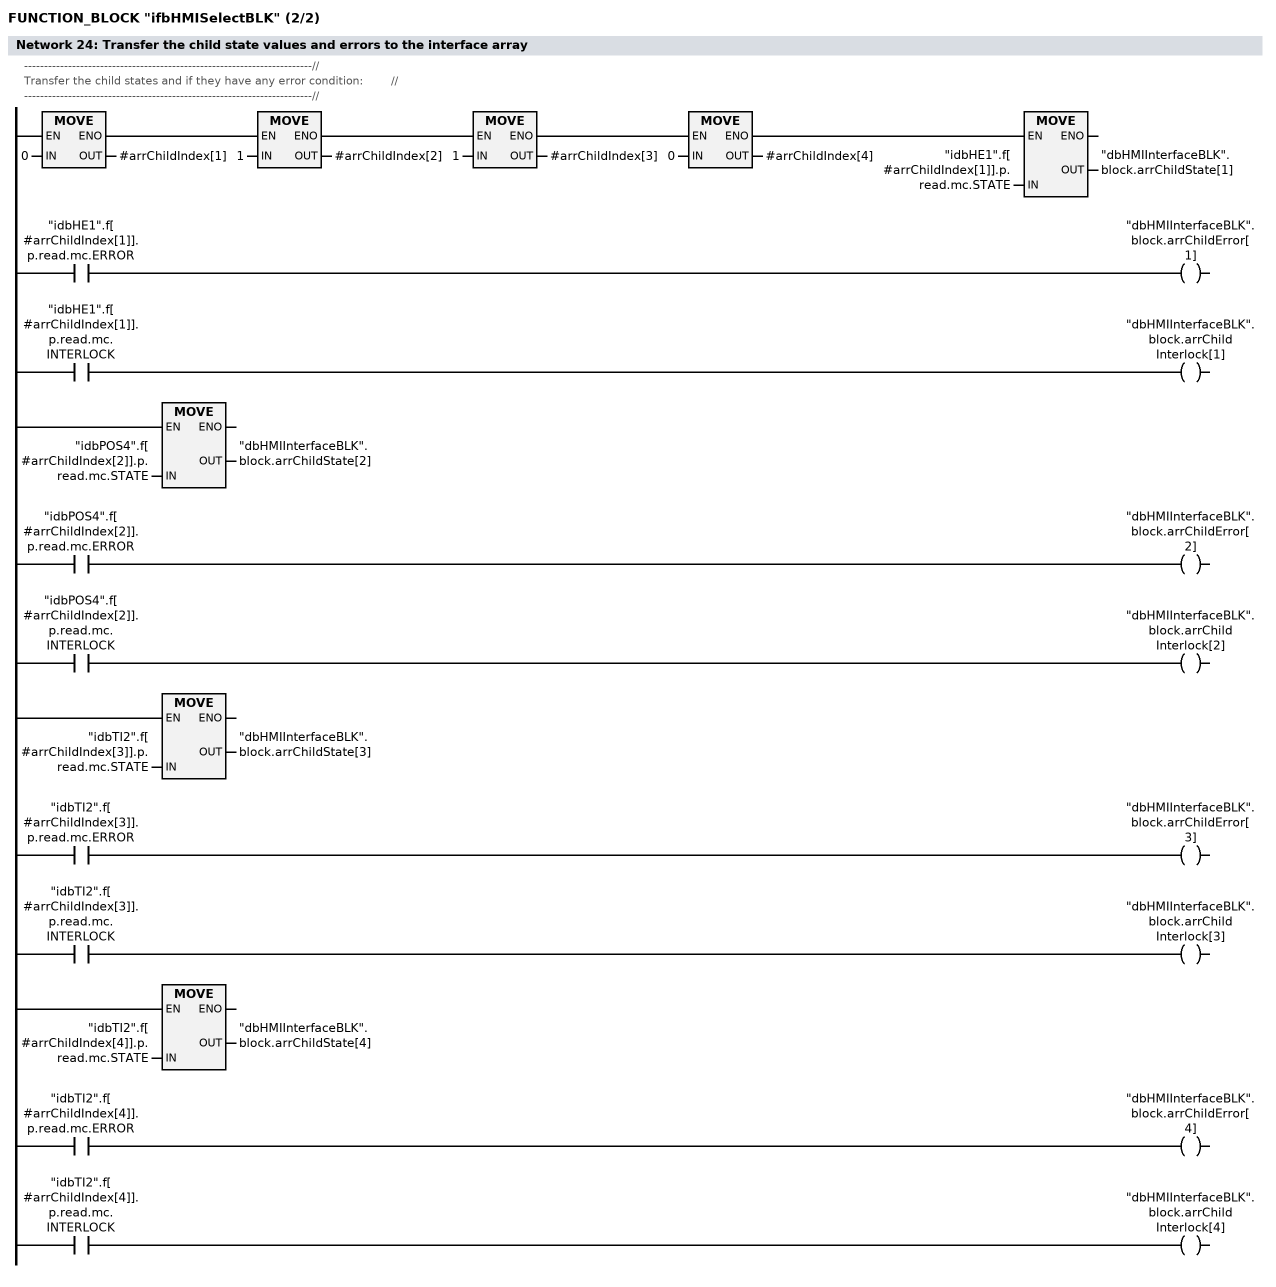
      L 0        ;// HE_FILTER HE1
      T #arrChildIndex[1];
      L 1        ;// POS_DRAIN POS4
      T #arrChildIndex[2];
      L 1        ;// TI_DRAIN TI2
      T #arrChildIndex[3];
      L 0        ;// TI_VENT TI2
      T #arrChildIndex[4];
      L "idbHE1".f[#arrChildIndex[1]].p.read.mc.STATE;
      T "dbHMIInterfaceBLK".block.arrChildState[1];
      A "idbHE1".f[#arrChildIndex[1]].p.read.mc.ERROR;
      = "dbHMIInterfaceBLK".block.arrChildError[1];
      A "idbHE1".f[#arrChildIndex[1]].p.read.mc.INTERLOCK;
      = "dbHMIInterfaceBLK".block.arrChildInterlock[1];
      L "idbPOS4".f[#arrChildIndex[2]].p.read.mc.STATE;
      T "dbHMIInterfaceBLK".block.arrChildState[2];
      A "idbPOS4".f[#arrChildIndex[2]].p.read.mc.ERROR;
      = "dbHMIInterfaceBLK".block.arrChildError[2];
      A "idbPOS4".f[#arrChildIndex[2]].p.read.mc.INTERLOCK;
      = "dbHMIInterfaceBLK".block.arrChildInterlock[2];
      L "idbTI2".f[#arrChildIndex[3]].p.read.mc.STATE;
      T "dbHMIInterfaceBLK".block.arrChildState[3];
      A "idbTI2".f[#arrChildIndex[3]].p.read.mc.ERROR;
      = "dbHMIInterfaceBLK".block.arrChildError[3];
      A "idbTI2".f[#arrChildIndex[3]].p.read.mc.INTERLOCK;
      = "dbHMIInterfaceBLK".block.arrChildInterlock[3];
      L "idbTI2".f[#arrChildIndex[4]].p.read.mc.STATE;
      T "dbHMIInterfaceBLK".block.arrChildState[4];
      A "idbTI2".f[#arrChildIndex[4]].p.read.mc.ERROR;
      = "dbHMIInterfaceBLK".block.arrChildError[4];
      A "idbTI2".f[#arrChildIndex[4]].p.read.mc.INTERLOCK;
      = "dbHMIInterfaceBLK".block.arrChildInterlock[4];

NETWORK
TITLE = Transfer the parameter values to the interface arrays
//------------------------------------------------------------------------//
// Transfer the parameter values:                                         //
//------------------------------------------------------------------------//
      AN "dbHMIInterfaceBLK".block.manual;
      JCN _manual_EG1005;
_manual_EG1005:      NOP 0;

NETWORK
TITLE = Transfer the parameter values to the interface arrays
//------------------------------------------------------------------------//
// Transfer the parameter values:                                         //
//------------------------------------------------------------------------//
      A "dbHMIInterfaceBLK".block.manual;
      JCN _auto_EG1005;
_auto_EG1005:      NOP 0;

_not_EG1005:      NOP 0;

NETWORK
TITLE = EG3005 S1 gas filter heating and drain valve and temperature indicator
//------------------------------------------------------------------------//
// Check if this BLK instance is selected:                                //
//------------------------------------------------------------------------//
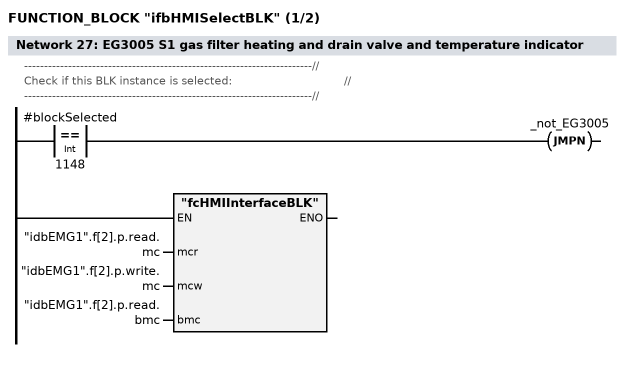
      A(;
      L #blockSelected;
      L 1148;
      ==I;
      );
      JCN _not_EG3005;

      CALL "fcHMIInterfaceBLK"
      (  mcr                         := "idbEMG1".f[2].p.read.mc ,
         mcw                         := "idbEMG1".f[2].p.write.mc ,
         bmc                         := "idbEMG1".f[2].p.read.bmc
      );

NETWORK
TITLE = Transfer the child state values and errors to the interface array
//------------------------------------------------------------------------//
// Transfer the child states and if they have any error condition:        //
//------------------------------------------------------------------------//
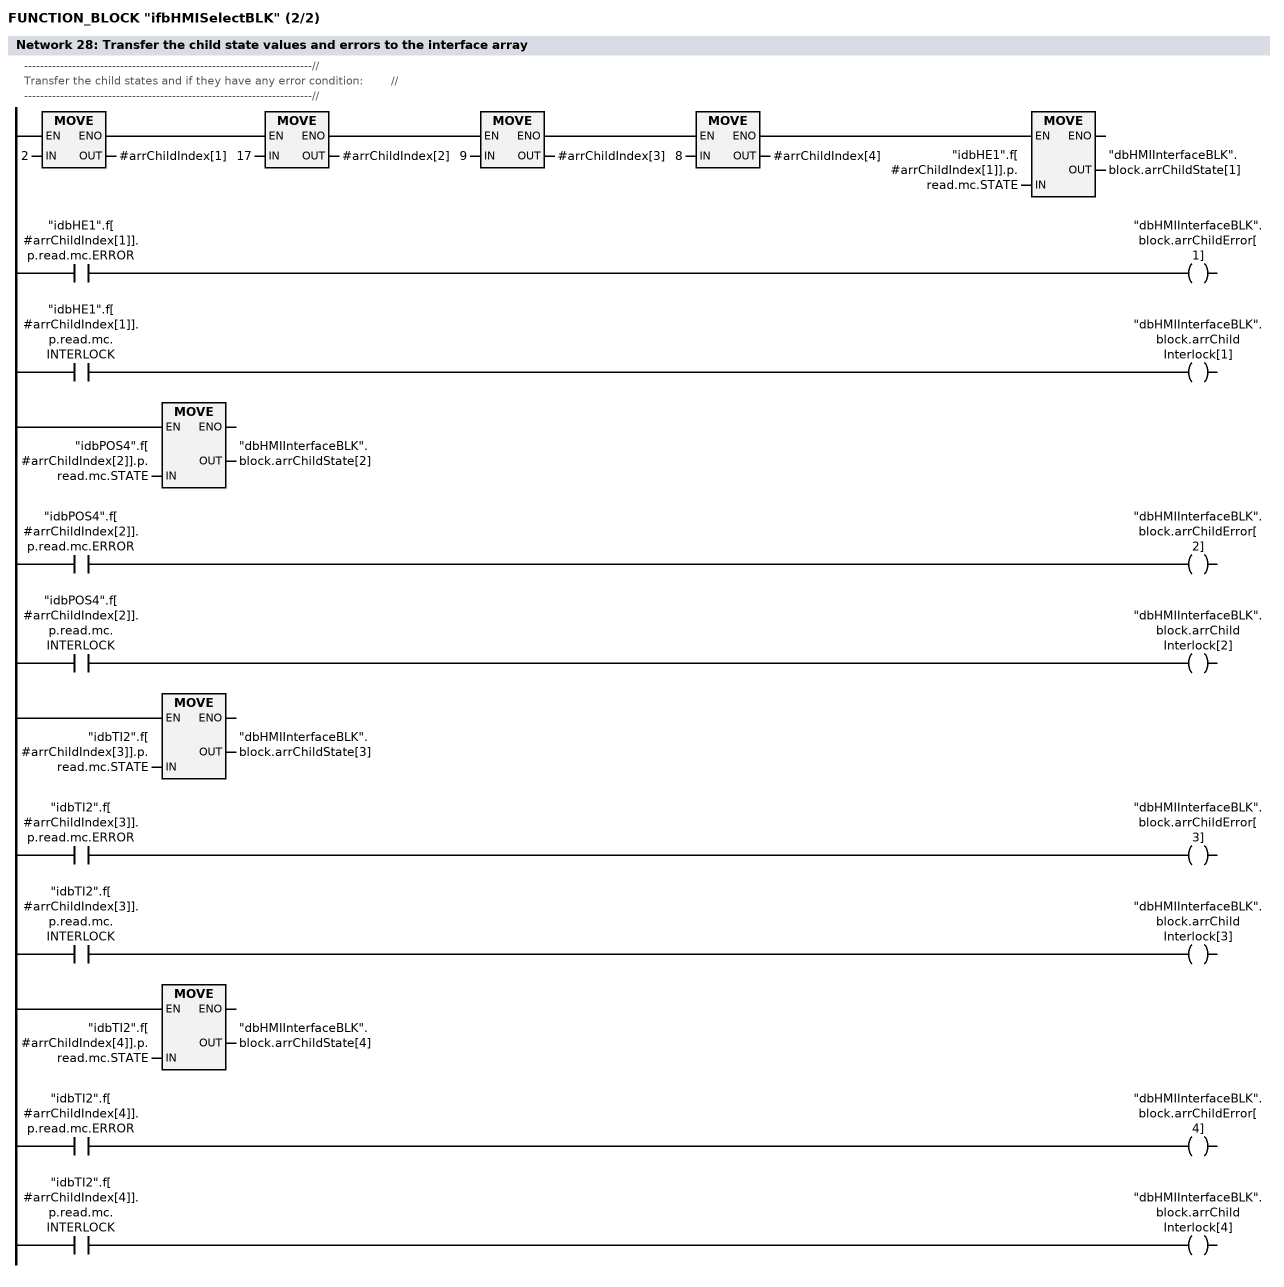
      L 2        ;// HE_FILTER HE1
      T #arrChildIndex[1];
      L 17        ;// POS_DRAIN POS4
      T #arrChildIndex[2];
      L 9        ;// TI_DRAIN TI2
      T #arrChildIndex[3];
      L 8        ;// TI_VENT TI2
      T #arrChildIndex[4];
      L "idbHE1".f[#arrChildIndex[1]].p.read.mc.STATE;
      T "dbHMIInterfaceBLK".block.arrChildState[1];
      A "idbHE1".f[#arrChildIndex[1]].p.read.mc.ERROR;
      = "dbHMIInterfaceBLK".block.arrChildError[1];
      A "idbHE1".f[#arrChildIndex[1]].p.read.mc.INTERLOCK;
      = "dbHMIInterfaceBLK".block.arrChildInterlock[1];
      L "idbPOS4".f[#arrChildIndex[2]].p.read.mc.STATE;
      T "dbHMIInterfaceBLK".block.arrChildState[2];
      A "idbPOS4".f[#arrChildIndex[2]].p.read.mc.ERROR;
      = "dbHMIInterfaceBLK".block.arrChildError[2];
      A "idbPOS4".f[#arrChildIndex[2]].p.read.mc.INTERLOCK;
      = "dbHMIInterfaceBLK".block.arrChildInterlock[2];
      L "idbTI2".f[#arrChildIndex[3]].p.read.mc.STATE;
      T "dbHMIInterfaceBLK".block.arrChildState[3];
      A "idbTI2".f[#arrChildIndex[3]].p.read.mc.ERROR;
      = "dbHMIInterfaceBLK".block.arrChildError[3];
      A "idbTI2".f[#arrChildIndex[3]].p.read.mc.INTERLOCK;
      = "dbHMIInterfaceBLK".block.arrChildInterlock[3];
      L "idbTI2".f[#arrChildIndex[4]].p.read.mc.STATE;
      T "dbHMIInterfaceBLK".block.arrChildState[4];
      A "idbTI2".f[#arrChildIndex[4]].p.read.mc.ERROR;
      = "dbHMIInterfaceBLK".block.arrChildError[4];
      A "idbTI2".f[#arrChildIndex[4]].p.read.mc.INTERLOCK;
      = "dbHMIInterfaceBLK".block.arrChildInterlock[4];

NETWORK
TITLE = Transfer the parameter values to the interface arrays
//------------------------------------------------------------------------//
// Transfer the parameter values:                                         //
//------------------------------------------------------------------------//
      AN "dbHMIInterfaceBLK".block.manual;
      JCN _manual_EG3005;
_manual_EG3005:      NOP 0;

NETWORK
TITLE = Transfer the parameter values to the interface arrays
//------------------------------------------------------------------------//
// Transfer the parameter values:                                         //
//------------------------------------------------------------------------//
      A "dbHMIInterfaceBLK".block.manual;
      JCN _auto_EG3005;
_auto_EG3005:      NOP 0;

_not_EG3005:      NOP 0;

NETWORK
TITLE = EM1009 M1 load cell
//------------------------------------------------------------------------//
// Check if this BLK instance is selected:                                //
//------------------------------------------------------------------------//
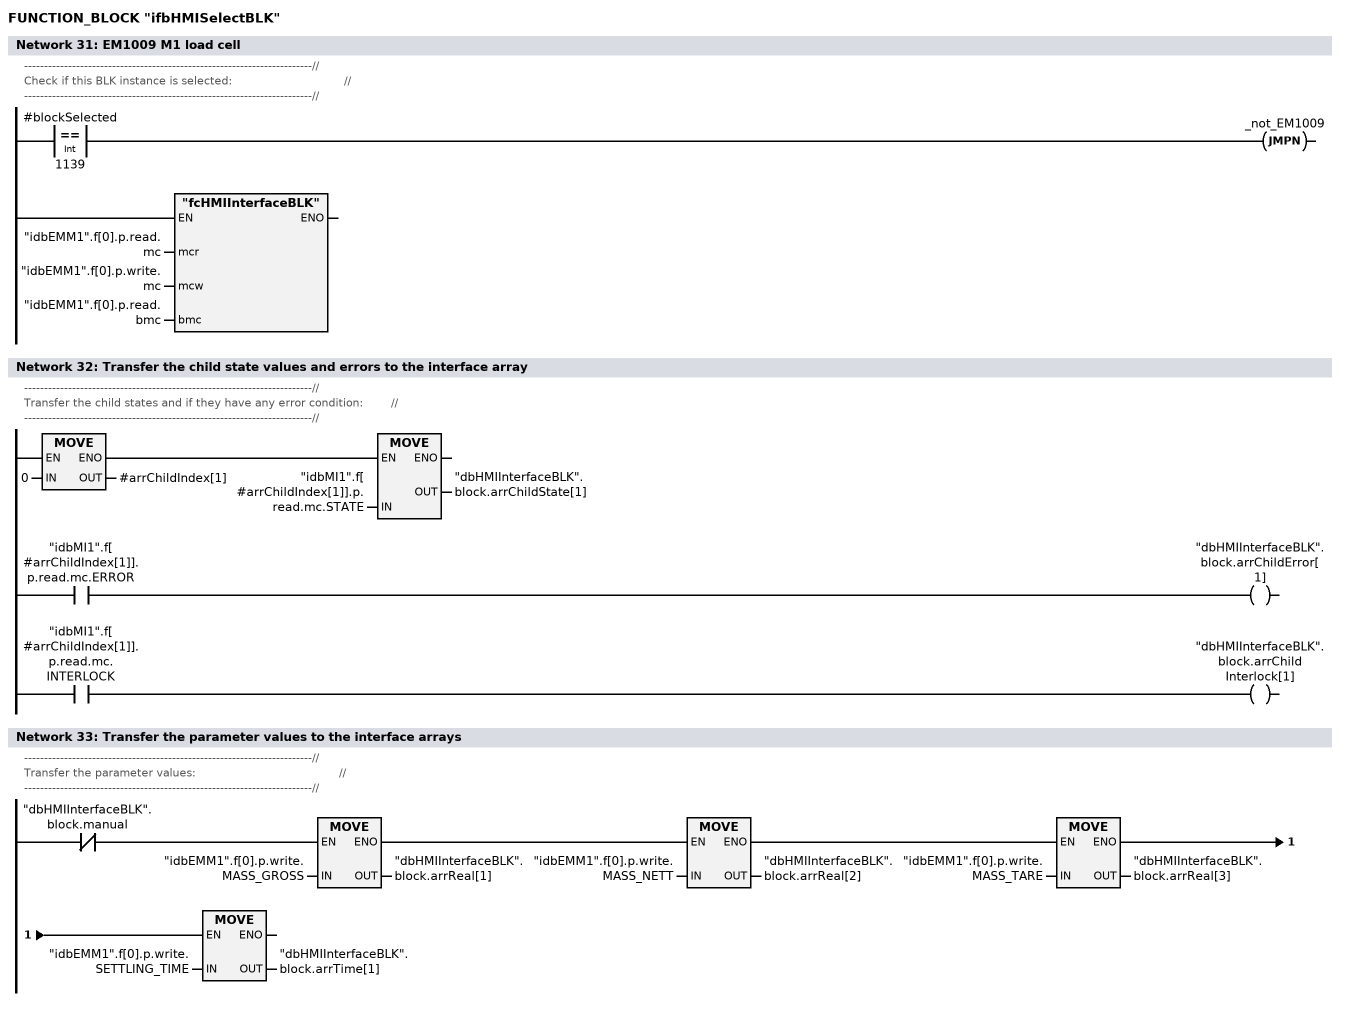
      A(;
      L #blockSelected;
      L 1139;
      ==I;
      );
      JCN _not_EM1009;

      CALL "fcHMIInterfaceBLK"
      (  mcr                         := "idbEMM1".f[0].p.read.mc ,
         mcw                         := "idbEMM1".f[0].p.write.mc ,
         bmc                         := "idbEMM1".f[0].p.read.bmc
      );

NETWORK
TITLE = Transfer the child state values and errors to the interface array
//------------------------------------------------------------------------//
// Transfer the child states and if they have any error condition:        //
//------------------------------------------------------------------------//
      L 0        ;// MI_VESSEL MI1
      T #arrChildIndex[1];
      L "idbMI1".f[#arrChildIndex[1]].p.read.mc.STATE;
      T "dbHMIInterfaceBLK".block.arrChildState[1];
      A "idbMI1".f[#arrChildIndex[1]].p.read.mc.ERROR;
      = "dbHMIInterfaceBLK".block.arrChildError[1];
      A "idbMI1".f[#arrChildIndex[1]].p.read.mc.INTERLOCK;
      = "dbHMIInterfaceBLK".block.arrChildInterlock[1];

NETWORK
TITLE = Transfer the parameter values to the interface arrays
//------------------------------------------------------------------------//
// Transfer the parameter values:                                         //
//------------------------------------------------------------------------//
      AN "dbHMIInterfaceBLK".block.manual;
      JCN _manual_EM1009;
      L "idbEMM1".f[0].p.write.MASS_GROSS;
      T "dbHMIInterfaceBLK".block.arrReal[1];
      L "idbEMM1".f[0].p.write.MASS_NETT;
      T "dbHMIInterfaceBLK".block.arrReal[2];
      L "idbEMM1".f[0].p.write.MASS_TARE;
      T "dbHMIInterfaceBLK".block.arrReal[3];
      L "idbEMM1".f[0].p.write.SETTLING_TIME;
      T "dbHMIInterfaceBLK".block.arrTime[1];
_manual_EM1009:      NOP 0;

NETWORK
TITLE = Transfer the parameter values to the interface arrays
//------------------------------------------------------------------------//
// Transfer the parameter values:                                         //
//------------------------------------------------------------------------//
      A "dbHMIInterfaceBLK".block.manual;
      JCN _auto_EM1009;
      L "dbHMIInterfaceBLK".block.arrReal[1];
      T "idbEMM1".f[0].p.write.MASS_GROSS;
      L "dbHMIInterfaceBLK".block.arrReal[2];
      T "idbEMM1".f[0].p.write.MASS_NETT;
      L "dbHMIInterfaceBLK".block.arrReal[3];
      T "idbEMM1".f[0].p.write.MASS_TARE;
      L "dbHMIInterfaceBLK".block.arrTime[1];
      T "idbEMM1".f[0].p.write.SETTLING_TIME;
_auto_EM1009:      NOP 0;

_not_EM1009:      NOP 0;

NETWORK
TITLE = ET1003 Manufacturing Filtration Line Heat Exchanger Temperature Control
//------------------------------------------------------------------------//
// Check if this BLK instance is selected:                                //
//------------------------------------------------------------------------//
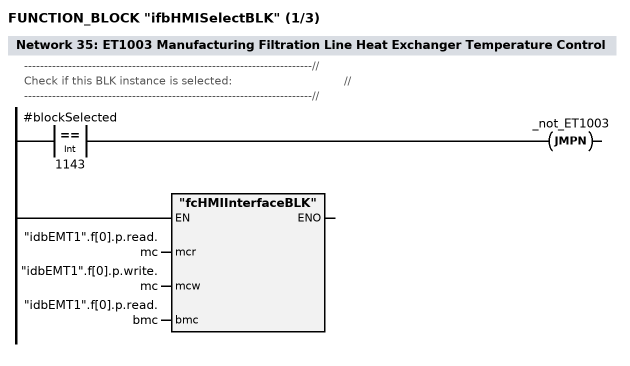
      A(;
      L #blockSelected;
      L 1143;
      ==I;
      );
      JCN _not_ET1003;

      CALL "fcHMIInterfaceBLK"
      (  mcr                         := "idbEMT1".f[0].p.read.mc ,
         mcw                         := "idbEMT1".f[0].p.write.mc ,
         bmc                         := "idbEMT1".f[0].p.read.bmc
      );

NETWORK
TITLE = Transfer the child state values and errors to the interface array
//------------------------------------------------------------------------//
// Transfer the child states and if they have any error condition:        //
//------------------------------------------------------------------------//
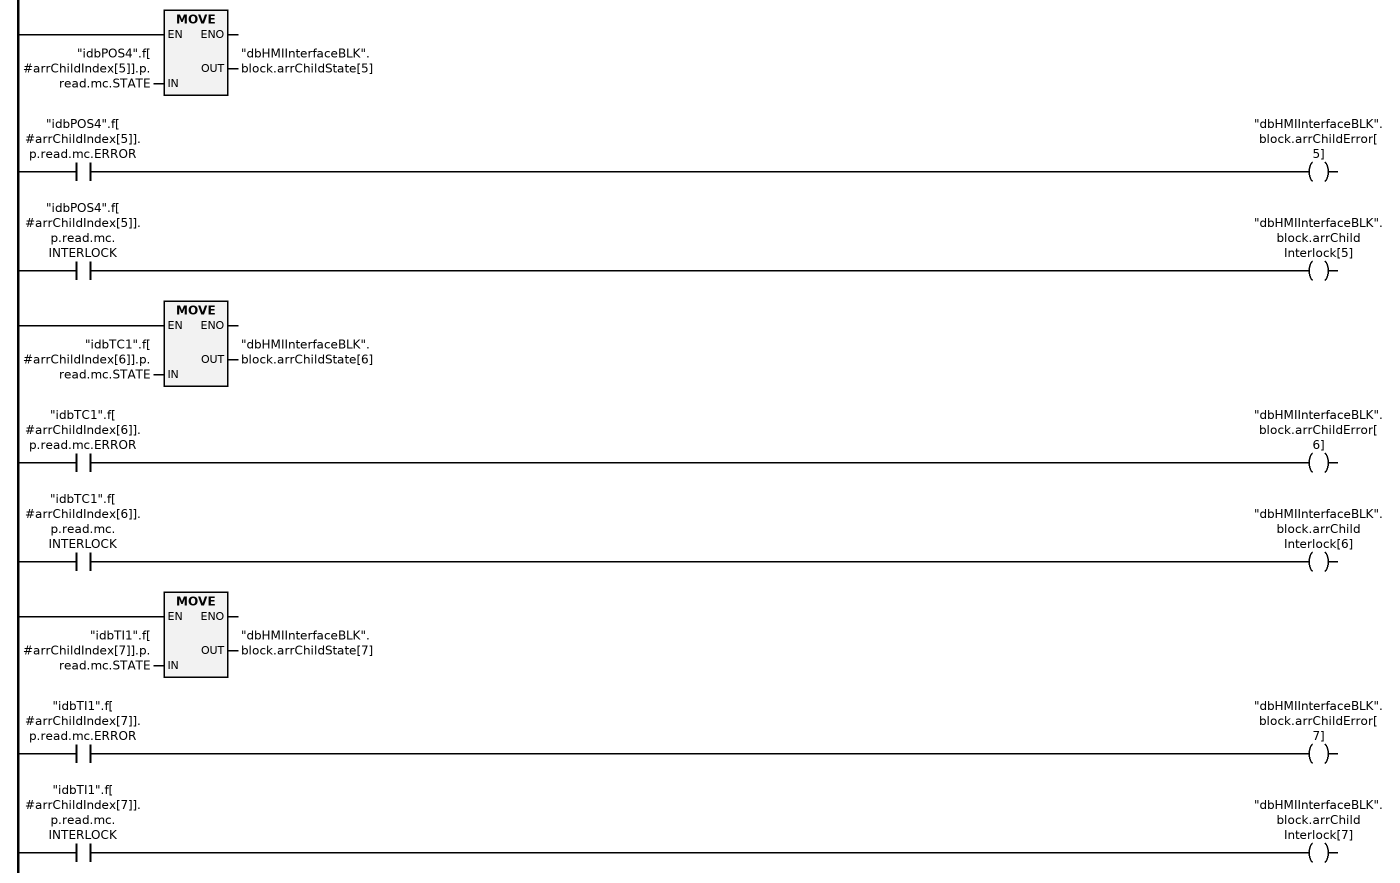
      L 0        ;// MOD_TCV MOD1
      T #arrChildIndex[1];
      L 25        ;// POS_RETURN POS4
      T #arrChildIndex[2];
      L 7        ;// POS_RETURNDRAIN POS4
      T #arrChildIndex[3];
      L 24        ;// POS_SUPPLY POS4
      T #arrChildIndex[4];
      L 6        ;// POS_SUPPLYDRAIN POS4
      T #arrChildIndex[5];
      L 0        ;// TC_HEX TC1
      T #arrChildIndex[6];
      L 1        ;// TI_HEX TI1
      T #arrChildIndex[7];
      L "idbMOD1".f[#arrChildIndex[1]].p.read.mc.STATE;
      T "dbHMIInterfaceBLK".block.arrChildState[1];
      A "idbMOD1".f[#arrChildIndex[1]].p.read.mc.ERROR;
      = "dbHMIInterfaceBLK".block.arrChildError[1];
      A "idbMOD1".f[#arrChildIndex[1]].p.read.mc.INTERLOCK;
      = "dbHMIInterfaceBLK".block.arrChildInterlock[1];
      L "idbPOS4".f[#arrChildIndex[2]].p.read.mc.STATE;
      T "dbHMIInterfaceBLK".block.arrChildState[2];
      A "idbPOS4".f[#arrChildIndex[2]].p.read.mc.ERROR;
      = "dbHMIInterfaceBLK".block.arrChildError[2];
      A "idbPOS4".f[#arrChildIndex[2]].p.read.mc.INTERLOCK;
      = "dbHMIInterfaceBLK".block.arrChildInterlock[2];
      L "idbPOS4".f[#arrChildIndex[3]].p.read.mc.STATE;
      T "dbHMIInterfaceBLK".block.arrChildState[3];
      A "idbPOS4".f[#arrChildIndex[3]].p.read.mc.ERROR;
      = "dbHMIInterfaceBLK".block.arrChildError[3];
      A "idbPOS4".f[#arrChildIndex[3]].p.read.mc.INTERLOCK;
      = "dbHMIInterfaceBLK".block.arrChildInterlock[3];
      L "idbPOS4".f[#arrChildIndex[4]].p.read.mc.STATE;
      T "dbHMIInterfaceBLK".block.arrChildState[4];
      A "idbPOS4".f[#arrChildIndex[4]].p.read.mc.ERROR;
      = "dbHMIInterfaceBLK".block.arrChildError[4];
      A "idbPOS4".f[#arrChildIndex[4]].p.read.mc.INTERLOCK;
      = "dbHMIInterfaceBLK".block.arrChildInterlock[4];
      L "idbPOS4".f[#arrChildIndex[5]].p.read.mc.STATE;
      T "dbHMIInterfaceBLK".block.arrChildState[5];
      A "idbPOS4".f[#arrChildIndex[5]].p.read.mc.ERROR;
      = "dbHMIInterfaceBLK".block.arrChildError[5];
      A "idbPOS4".f[#arrChildIndex[5]].p.read.mc.INTERLOCK;
      = "dbHMIInterfaceBLK".block.arrChildInterlock[5];
      L "idbTC1".f[#arrChildIndex[6]].p.read.mc.STATE;
      T "dbHMIInterfaceBLK".block.arrChildState[6];
      A "idbTC1".f[#arrChildIndex[6]].p.read.mc.ERROR;
      = "dbHMIInterfaceBLK".block.arrChildError[6];
      A "idbTC1".f[#arrChildIndex[6]].p.read.mc.INTERLOCK;
      = "dbHMIInterfaceBLK".block.arrChildInterlock[6];
      L "idbTI1".f[#arrChildIndex[7]].p.read.mc.STATE;
      T "dbHMIInterfaceBLK".block.arrChildState[7];
      A "idbTI1".f[#arrChildIndex[7]].p.read.mc.ERROR;
      = "dbHMIInterfaceBLK".block.arrChildError[7];
      A "idbTI1".f[#arrChildIndex[7]].p.read.mc.INTERLOCK;
      = "dbHMIInterfaceBLK".block.arrChildInterlock[7];

NETWORK
TITLE = Transfer the parameter values to the interface arrays
//------------------------------------------------------------------------//
// Transfer the parameter values:                                         //
//------------------------------------------------------------------------//
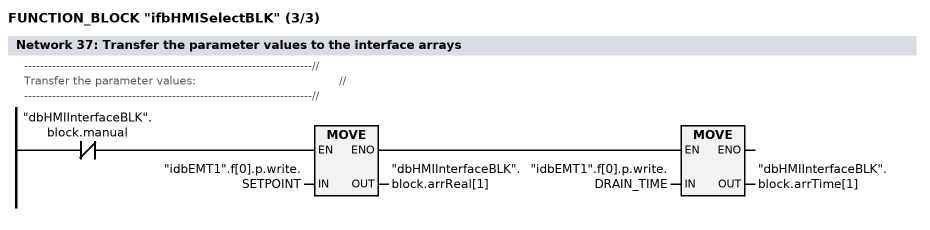
      AN "dbHMIInterfaceBLK".block.manual;
      JCN _manual_ET1003;
      L "idbEMT1".f[0].p.write.SETPOINT;
      T "dbHMIInterfaceBLK".block.arrReal[1];
      L "idbEMT1".f[0].p.write.DRAIN_TIME;
      T "dbHMIInterfaceBLK".block.arrTime[1];
_manual_ET1003:      NOP 0;

NETWORK
TITLE = Transfer the parameter values to the interface arrays
//------------------------------------------------------------------------//
// Transfer the parameter values:                                         //
//------------------------------------------------------------------------//
      A "dbHMIInterfaceBLK".block.manual;
      JCN _auto_ET1003;
      L "dbHMIInterfaceBLK".block.arrReal[1];
      T "idbEMT1".f[0].p.write.SETPOINT;
      L "dbHMIInterfaceBLK".block.arrTime[1];
      T "idbEMT1".f[0].p.write.DRAIN_TIME;
_auto_ET1003:      NOP 0;

_not_ET1003:      NOP 0;

NETWORK
TITLE = EV1004 M1 vessel mounted equipment and valves
//------------------------------------------------------------------------//
// Check if this BLK instance is selected:                                //
//------------------------------------------------------------------------//
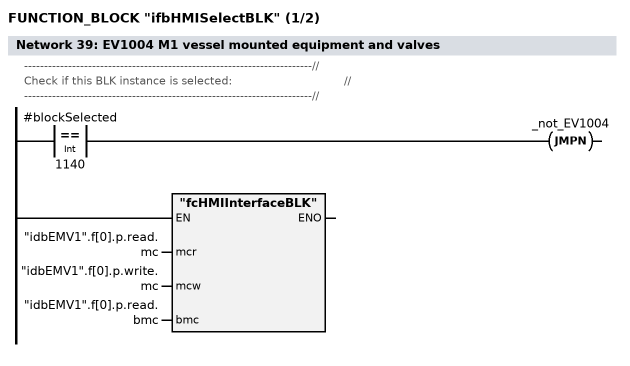
      A(;
      L #blockSelected;
      L 1140;
      ==I;
      );
      JCN _not_EV1004;

      CALL "fcHMIInterfaceBLK"
      (  mcr                         := "idbEMV1".f[0].p.read.mc ,
         mcw                         := "idbEMV1".f[0].p.write.mc ,
         bmc                         := "idbEMV1".f[0].p.read.bmc
      );

NETWORK
TITLE = Transfer the child state values and errors to the interface array
//------------------------------------------------------------------------//
// Transfer the child states and if they have any error condition:        //
//------------------------------------------------------------------------//
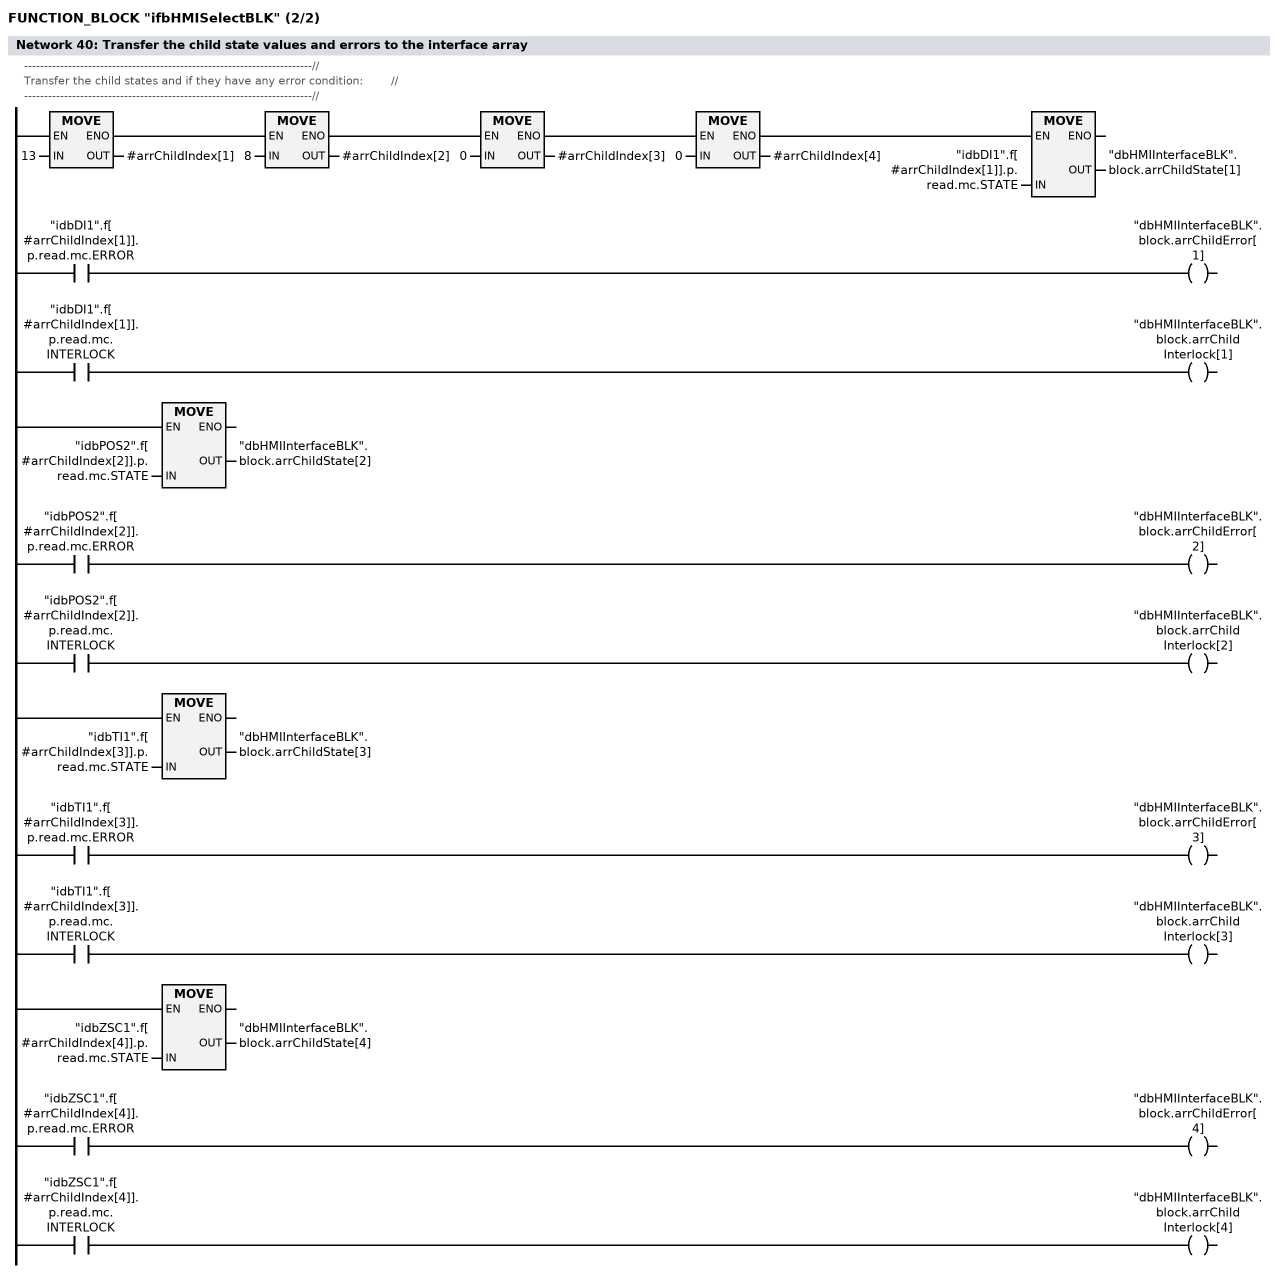
      L 13        ;// DI_BURST DI1
      T #arrChildIndex[1];
      L 8        ;// POS_OUTLET POS2
      T #arrChildIndex[2];
      L 0        ;// TI_VESSEL TI1
      T #arrChildIndex[3];
      L 0        ;// ZSC_MANWAY ZSC1
      T #arrChildIndex[4];
      L "idbDI1".f[#arrChildIndex[1]].p.read.mc.STATE;
      T "dbHMIInterfaceBLK".block.arrChildState[1];
      A "idbDI1".f[#arrChildIndex[1]].p.read.mc.ERROR;
      = "dbHMIInterfaceBLK".block.arrChildError[1];
      A "idbDI1".f[#arrChildIndex[1]].p.read.mc.INTERLOCK;
      = "dbHMIInterfaceBLK".block.arrChildInterlock[1];
      L "idbPOS2".f[#arrChildIndex[2]].p.read.mc.STATE;
      T "dbHMIInterfaceBLK".block.arrChildState[2];
      A "idbPOS2".f[#arrChildIndex[2]].p.read.mc.ERROR;
      = "dbHMIInterfaceBLK".block.arrChildError[2];
      A "idbPOS2".f[#arrChildIndex[2]].p.read.mc.INTERLOCK;
      = "dbHMIInterfaceBLK".block.arrChildInterlock[2];
      L "idbTI1".f[#arrChildIndex[3]].p.read.mc.STATE;
      T "dbHMIInterfaceBLK".block.arrChildState[3];
      A "idbTI1".f[#arrChildIndex[3]].p.read.mc.ERROR;
      = "dbHMIInterfaceBLK".block.arrChildError[3];
      A "idbTI1".f[#arrChildIndex[3]].p.read.mc.INTERLOCK;
      = "dbHMIInterfaceBLK".block.arrChildInterlock[3];
      L "idbZSC1".f[#arrChildIndex[4]].p.read.mc.STATE;
      T "dbHMIInterfaceBLK".block.arrChildState[4];
      A "idbZSC1".f[#arrChildIndex[4]].p.read.mc.ERROR;
      = "dbHMIInterfaceBLK".block.arrChildError[4];
      A "idbZSC1".f[#arrChildIndex[4]].p.read.mc.INTERLOCK;
      = "dbHMIInterfaceBLK".block.arrChildInterlock[4];

NETWORK
TITLE = Transfer the parameter values to the interface arrays
//------------------------------------------------------------------------//
// Transfer the parameter values:                                         //
//------------------------------------------------------------------------//
      AN "dbHMIInterfaceBLK".block.manual;
      JCN _manual_EV1004;
_manual_EV1004:      NOP 0;

NETWORK
TITLE = Transfer the parameter values to the interface arrays
//------------------------------------------------------------------------//
// Transfer the parameter values:                                         //
//------------------------------------------------------------------------//
      A "dbHMIInterfaceBLK".block.manual;
      JCN _auto_EV1004;
_auto_EV1004:      NOP 0;

_not_EV1004:      NOP 0;

NETWORK
TITLE = EV1008 M1 Vessel Inlet Connection
//------------------------------------------------------------------------//
// Check if this BLK instance is selected:                                //
//------------------------------------------------------------------------//
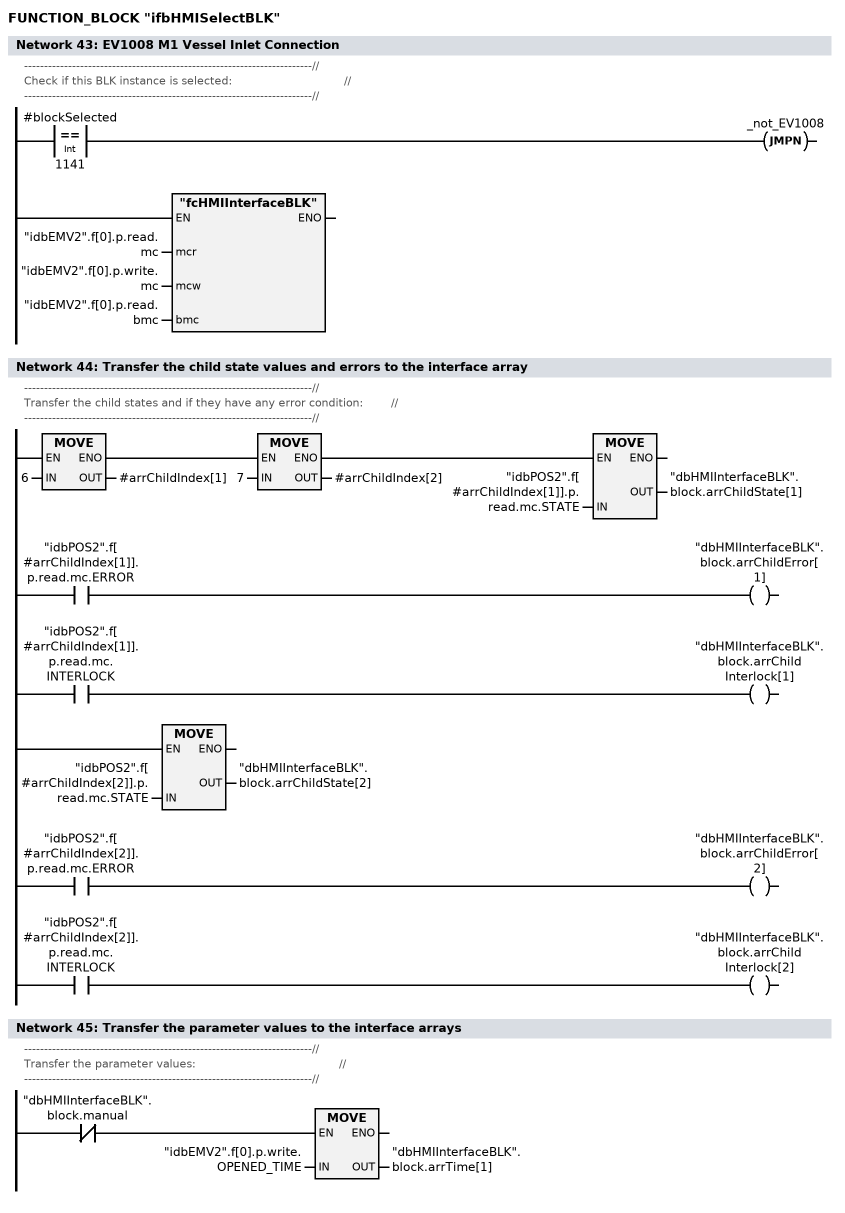
      A(;
      L #blockSelected;
      L 1141;
      ==I;
      );
      JCN _not_EV1008;

      CALL "fcHMIInterfaceBLK"
      (  mcr                         := "idbEMV2".f[0].p.read.mc ,
         mcw                         := "idbEMV2".f[0].p.write.mc ,
         bmc                         := "idbEMV2".f[0].p.read.bmc
      );

NETWORK
TITLE = Transfer the child state values and errors to the interface array
//------------------------------------------------------------------------//
// Transfer the child states and if they have any error condition:        //
//------------------------------------------------------------------------//
      L 6        ;// POS_SPRAYBALL1 POS2
      T #arrChildIndex[1];
      L 7        ;// POS_SPRAYBALL2 POS2
      T #arrChildIndex[2];
      L "idbPOS2".f[#arrChildIndex[1]].p.read.mc.STATE;
      T "dbHMIInterfaceBLK".block.arrChildState[1];
      A "idbPOS2".f[#arrChildIndex[1]].p.read.mc.ERROR;
      = "dbHMIInterfaceBLK".block.arrChildError[1];
      A "idbPOS2".f[#arrChildIndex[1]].p.read.mc.INTERLOCK;
      = "dbHMIInterfaceBLK".block.arrChildInterlock[1];
      L "idbPOS2".f[#arrChildIndex[2]].p.read.mc.STATE;
      T "dbHMIInterfaceBLK".block.arrChildState[2];
      A "idbPOS2".f[#arrChildIndex[2]].p.read.mc.ERROR;
      = "dbHMIInterfaceBLK".block.arrChildError[2];
      A "idbPOS2".f[#arrChildIndex[2]].p.read.mc.INTERLOCK;
      = "dbHMIInterfaceBLK".block.arrChildInterlock[2];

NETWORK
TITLE = Transfer the parameter values to the interface arrays
//------------------------------------------------------------------------//
// Transfer the parameter values:                                         //
//------------------------------------------------------------------------//
      AN "dbHMIInterfaceBLK".block.manual;
      JCN _manual_EV1008;
      L "idbEMV2".f[0].p.write.OPENED_TIME;
      T "dbHMIInterfaceBLK".block.arrTime[1];
_manual_EV1008:      NOP 0;

NETWORK
TITLE = Transfer the parameter values to the interface arrays
//------------------------------------------------------------------------//
// Transfer the parameter values:                                         //
//------------------------------------------------------------------------//
      A "dbHMIInterfaceBLK".block.manual;
      JCN _auto_EV1008;
      L "dbHMIInterfaceBLK".block.arrTime[1];
      T "idbEMV2".f[0].p.write.OPENED_TIME;
_auto_EV1008:      NOP 0;

_not_EV1008:      NOP 0;

NETWORK
TITLE = EV3004 S1 vessel mounted equipment and valves
//------------------------------------------------------------------------//
// Check if this BLK instance is selected:                                //
//------------------------------------------------------------------------//
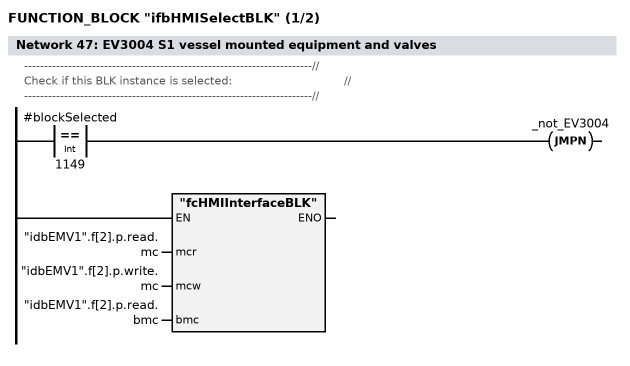
      A(;
      L #blockSelected;
      L 1149;
      ==I;
      );
      JCN _not_EV3004;

      CALL "fcHMIInterfaceBLK"
      (  mcr                         := "idbEMV1".f[2].p.read.mc ,
         mcw                         := "idbEMV1".f[2].p.write.mc ,
         bmc                         := "idbEMV1".f[2].p.read.bmc
      );

NETWORK
TITLE = Transfer the child state values and errors to the interface array
//------------------------------------------------------------------------//
// Transfer the child states and if they have any error condition:        //
//------------------------------------------------------------------------//
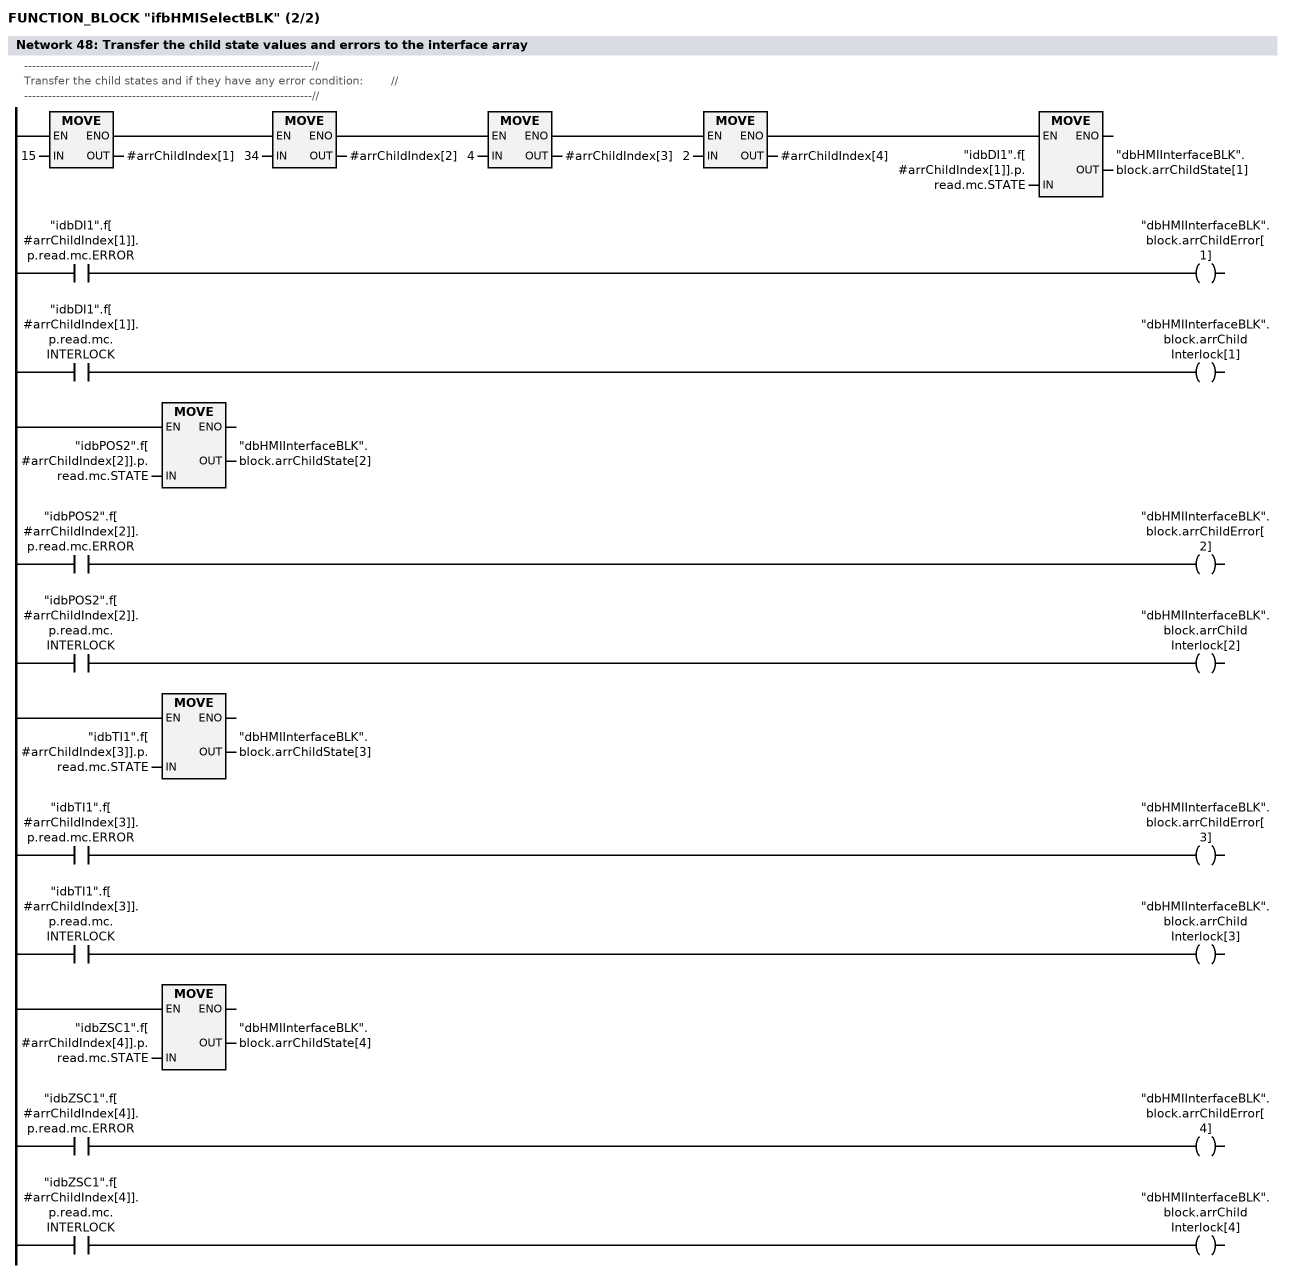
      L 15        ;// DI_BURST DI1
      T #arrChildIndex[1];
      L 34        ;// POS_OUTLET POS2
      T #arrChildIndex[2];
      L 4        ;// TI_VESSEL TI1
      T #arrChildIndex[3];
      L 2        ;// ZSC_MANWAY ZSC1
      T #arrChildIndex[4];
      L "idbDI1".f[#arrChildIndex[1]].p.read.mc.STATE;
      T "dbHMIInterfaceBLK".block.arrChildState[1];
      A "idbDI1".f[#arrChildIndex[1]].p.read.mc.ERROR;
      = "dbHMIInterfaceBLK".block.arrChildError[1];
      A "idbDI1".f[#arrChildIndex[1]].p.read.mc.INTERLOCK;
      = "dbHMIInterfaceBLK".block.arrChildInterlock[1];
      L "idbPOS2".f[#arrChildIndex[2]].p.read.mc.STATE;
      T "dbHMIInterfaceBLK".block.arrChildState[2];
      A "idbPOS2".f[#arrChildIndex[2]].p.read.mc.ERROR;
      = "dbHMIInterfaceBLK".block.arrChildError[2];
      A "idbPOS2".f[#arrChildIndex[2]].p.read.mc.INTERLOCK;
      = "dbHMIInterfaceBLK".block.arrChildInterlock[2];
      L "idbTI1".f[#arrChildIndex[3]].p.read.mc.STATE;
      T "dbHMIInterfaceBLK".block.arrChildState[3];
      A "idbTI1".f[#arrChildIndex[3]].p.read.mc.ERROR;
      = "dbHMIInterfaceBLK".block.arrChildError[3];
      A "idbTI1".f[#arrChildIndex[3]].p.read.mc.INTERLOCK;
      = "dbHMIInterfaceBLK".block.arrChildInterlock[3];
      L "idbZSC1".f[#arrChildIndex[4]].p.read.mc.STATE;
      T "dbHMIInterfaceBLK".block.arrChildState[4];
      A "idbZSC1".f[#arrChildIndex[4]].p.read.mc.ERROR;
      = "dbHMIInterfaceBLK".block.arrChildError[4];
      A "idbZSC1".f[#arrChildIndex[4]].p.read.mc.INTERLOCK;
      = "dbHMIInterfaceBLK".block.arrChildInterlock[4];

NETWORK
TITLE = Transfer the parameter values to the interface arrays
//------------------------------------------------------------------------//
// Transfer the parameter values:                                         //
//------------------------------------------------------------------------//
      AN "dbHMIInterfaceBLK".block.manual;
      JCN _manual_EV3004;
_manual_EV3004:      NOP 0;

NETWORK
TITLE = Transfer the parameter values to the interface arrays
//------------------------------------------------------------------------//
// Transfer the parameter values:                                         //
//------------------------------------------------------------------------//
      A "dbHMIInterfaceBLK".block.manual;
      JCN _auto_EV3004;
_auto_EV3004:      NOP 0;

_not_EV3004:      NOP 0;

NETWORK
TITLE = EV3008 S1 Vessel Inlet Connection
//------------------------------------------------------------------------//
// Check if this BLK instance is selected:                                //
//------------------------------------------------------------------------//
